// TIA Portal V18 export
FUNCTION_BLOCK "ST10_Flow8_FRobot_2"   // FB1078, GRAPH
// stored: AcknowledgeErrorsRequired false, AutoNumber false, GraphVersion 6.0, InitialValuesAcquisition false, SetENOAutomatically false
   // inherited from GRAPH_BASE
   VAR_INPUT
      INIT_SQ { ExternalAccessible := 'False'; ExternalVisible := 'False'; ExternalWritable := 'False'} : Bool := false;   // Set sequence to initial state
      iSysInface : "RCS_SysComInterface_V1";
   END_VAR
   VAR_IN_OUT
      ioPM_Inface : "RCS_PMInterface_V1";
      ioStatus : Int;
      Auto_Run_after_NG_box_closed : Bool;
   END_VAR
   VAR
      sCtrlMode { S7_SetPoint := 'True'} : "SysFlowCtrlGraph";
      sUpdMES_Data : Bool;   // 更新MES数据
      工件放行中 : Bool;
      前站站号 { ExternalAccessible := 'False'; ExternalVisible := 'False'; ExternalWritable := 'False'} : UInt;
      本站站号 { ExternalAccessible := 'False'; ExternalVisible := 'False'; ExternalWritable := 'False'} : UInt;
      弹窗Temp : Array[1..10] of Int;
      AlarmID : Int;
      TON { S7_SetPoint := 'True'} : Array[0..10] of TON_TIME;
      TOF { S7_SetPoint := 'True'} : Array[0..10] of TOF_TIME;
      sUP { S7_SetPoint := 'True'} : Array[0..10] of Bool;
      更新RFID完成 : Bool;
   END_VAR
   VAR_TEMP
      Tempresult : USInt;
      本站站号乘10 : UInt;
   END_VAR
   VAR CONSTANT
      Gripper_empty : Int := 0;
      "Gripper_have_OK_part_NO-MES" : Int := 199;
      Gripper_have_OK_part : Int := 110;
      Gripper_have_uknown_part : Int := 100;
      Gripper_Product_DMC_not_readable : Int := 155;
   END_VAR
   // // TON[0] : 托盘流入1托盘到位传感器
   // // TON[1] : 托盘流入1托盘到位传感器
   // // TON[2] : 托盘流入1产品有无传感器
   // // TON[3] : 托盘流入1产品有无传感器
   // // TON[4] : 托盘流入1姿态检测光电2
   // // TON[5] : 托盘流入1姿态检测光电3
   // // TON[0].Q : 托盘流入1托盘到位
   // // TON[1].Q : 托盘流入1托盘无
   // // TON[2].Q : 托盘流入1有产品
   // // TON[3].Q : 托盘流入1无产品
   // // TON[4].Q : 托盘流入1姿态检测光电2
   // // TON[5].Q : 托盘流入1姿态检测光电3
BEGIN
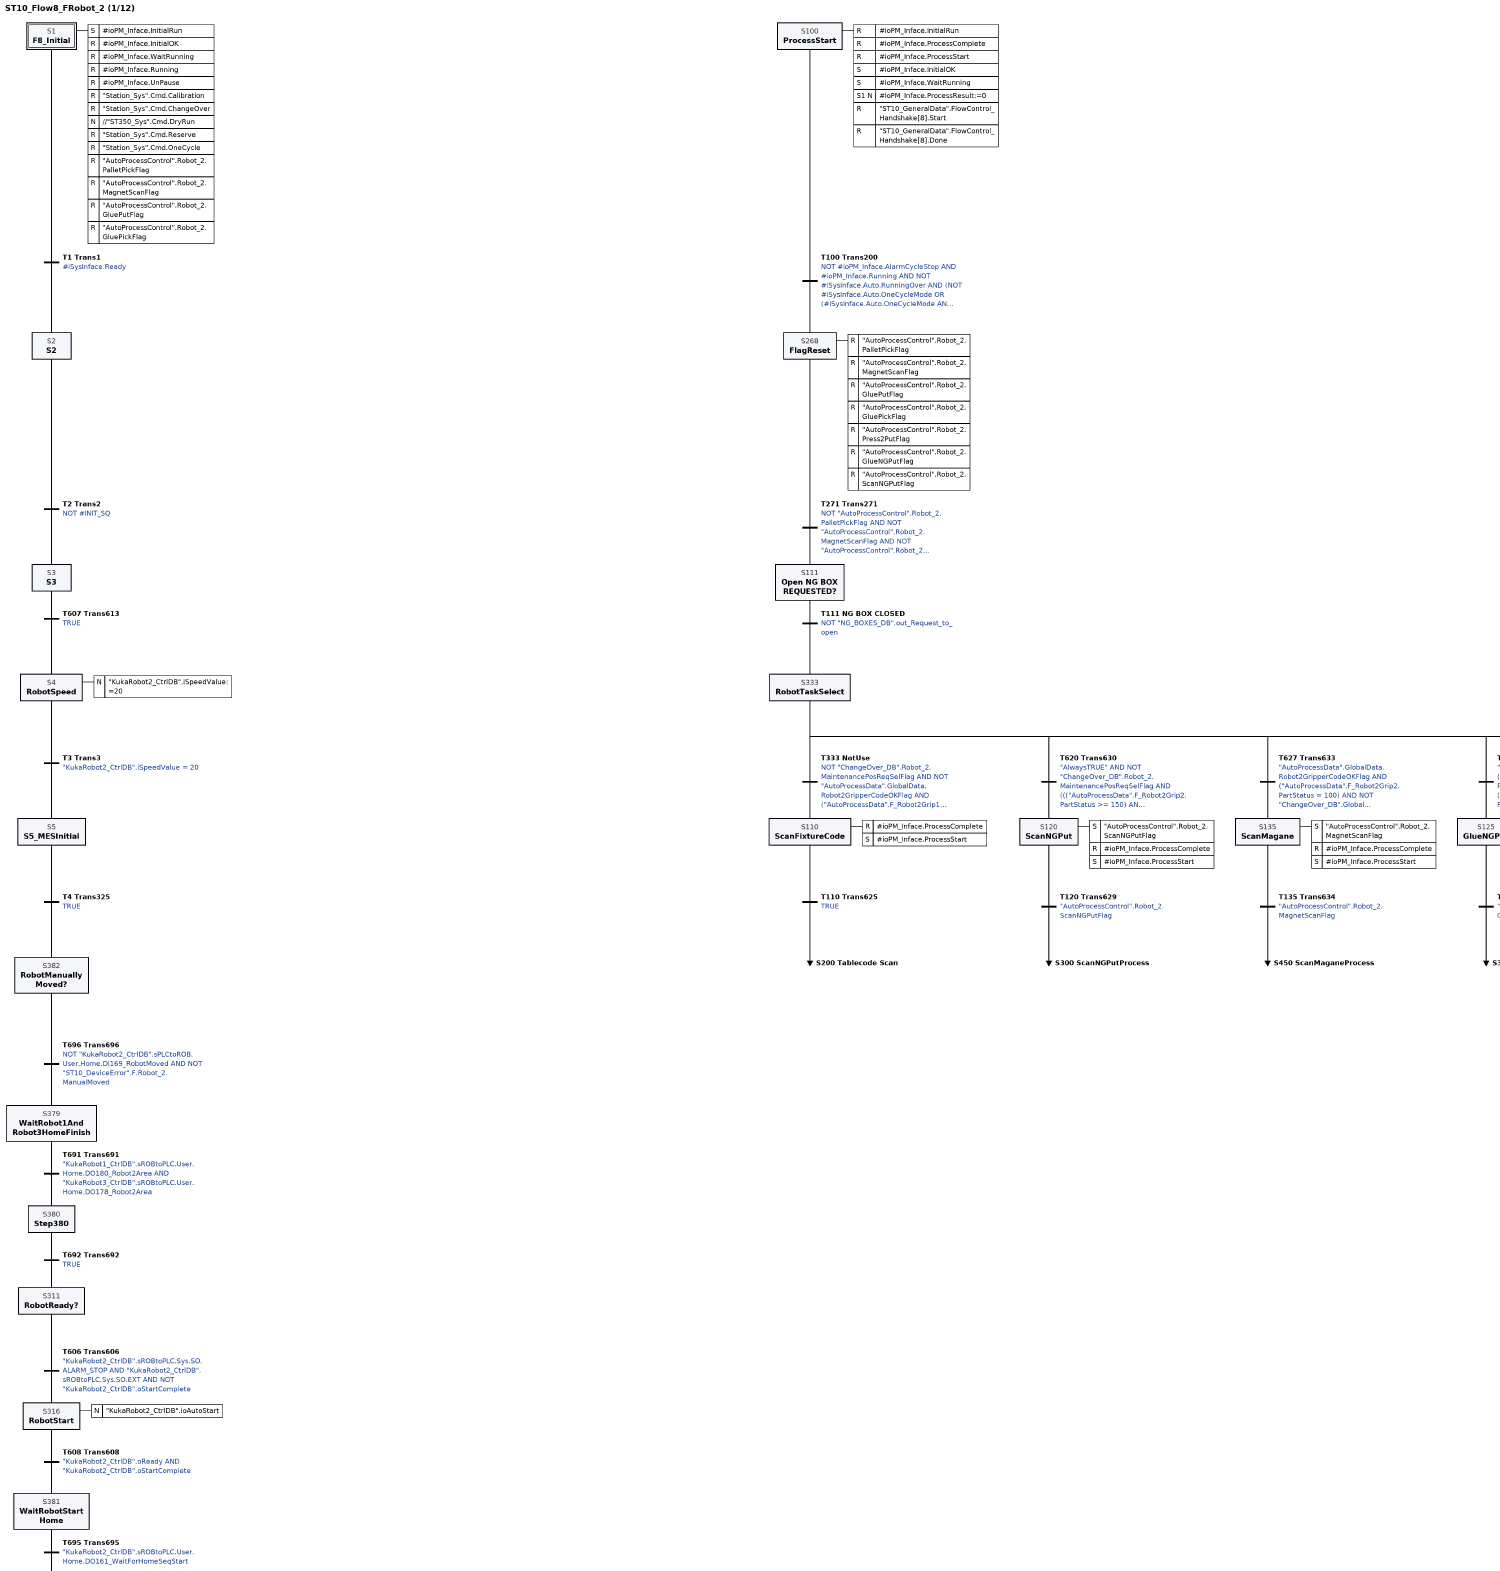
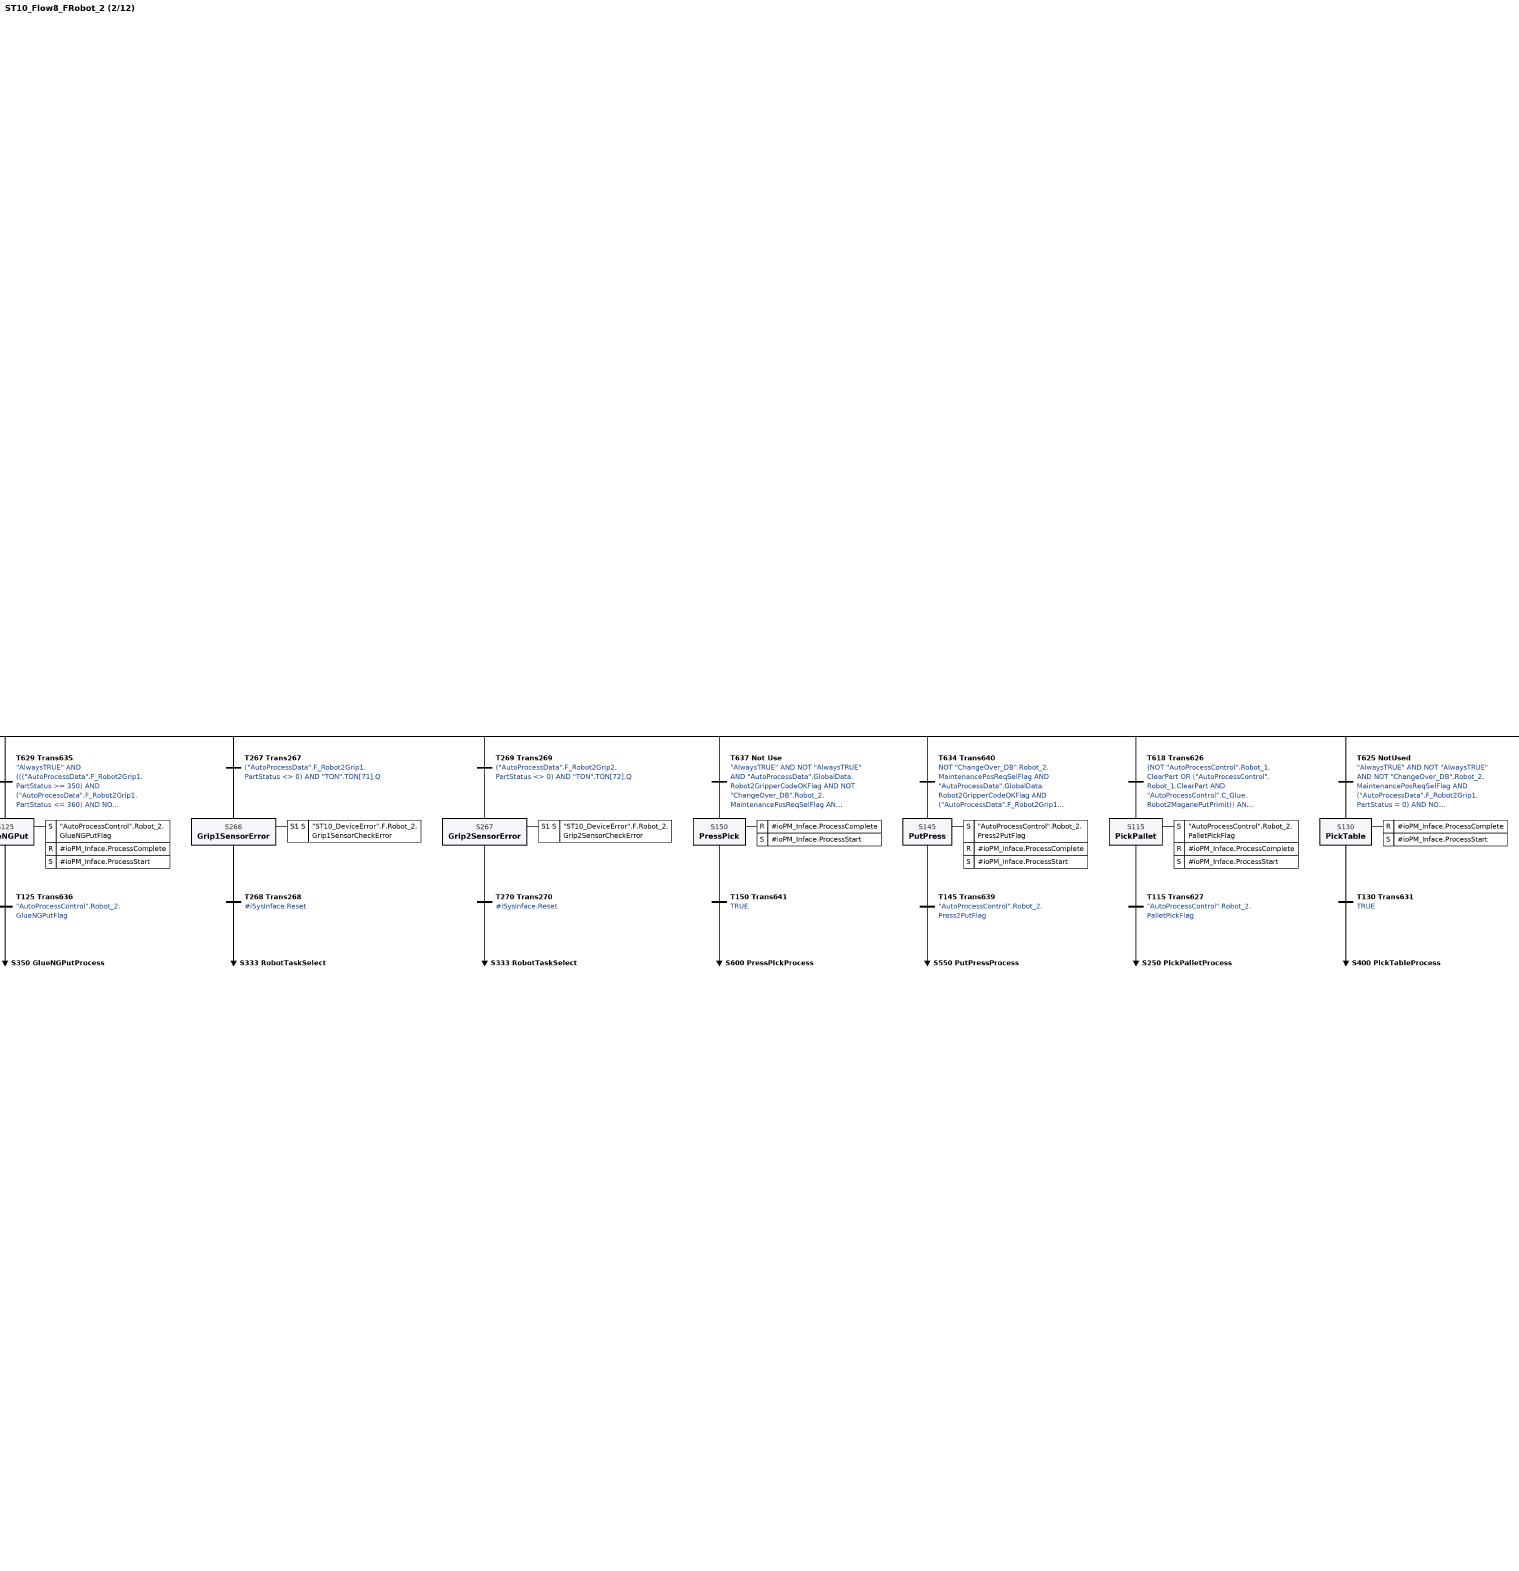
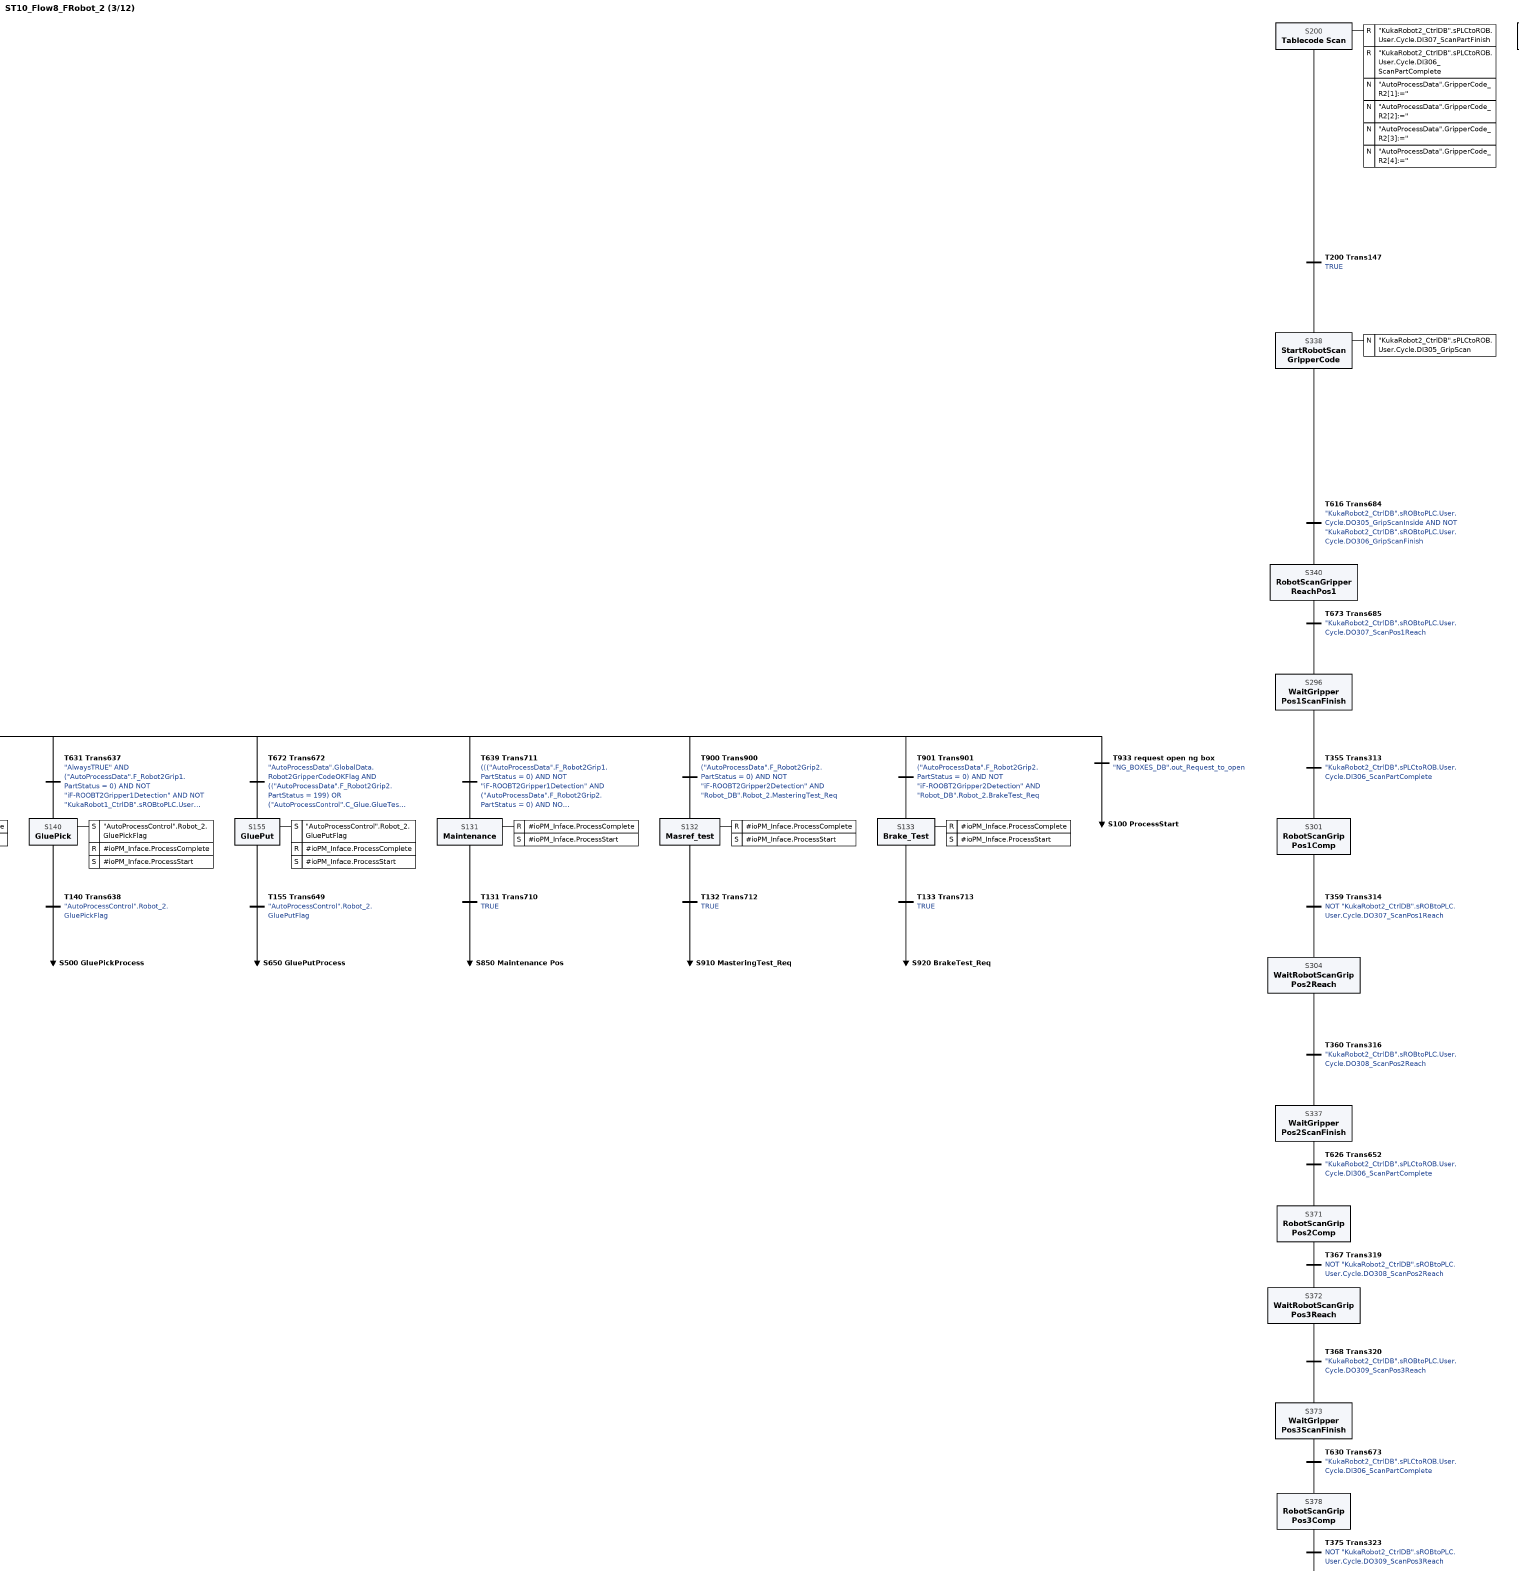
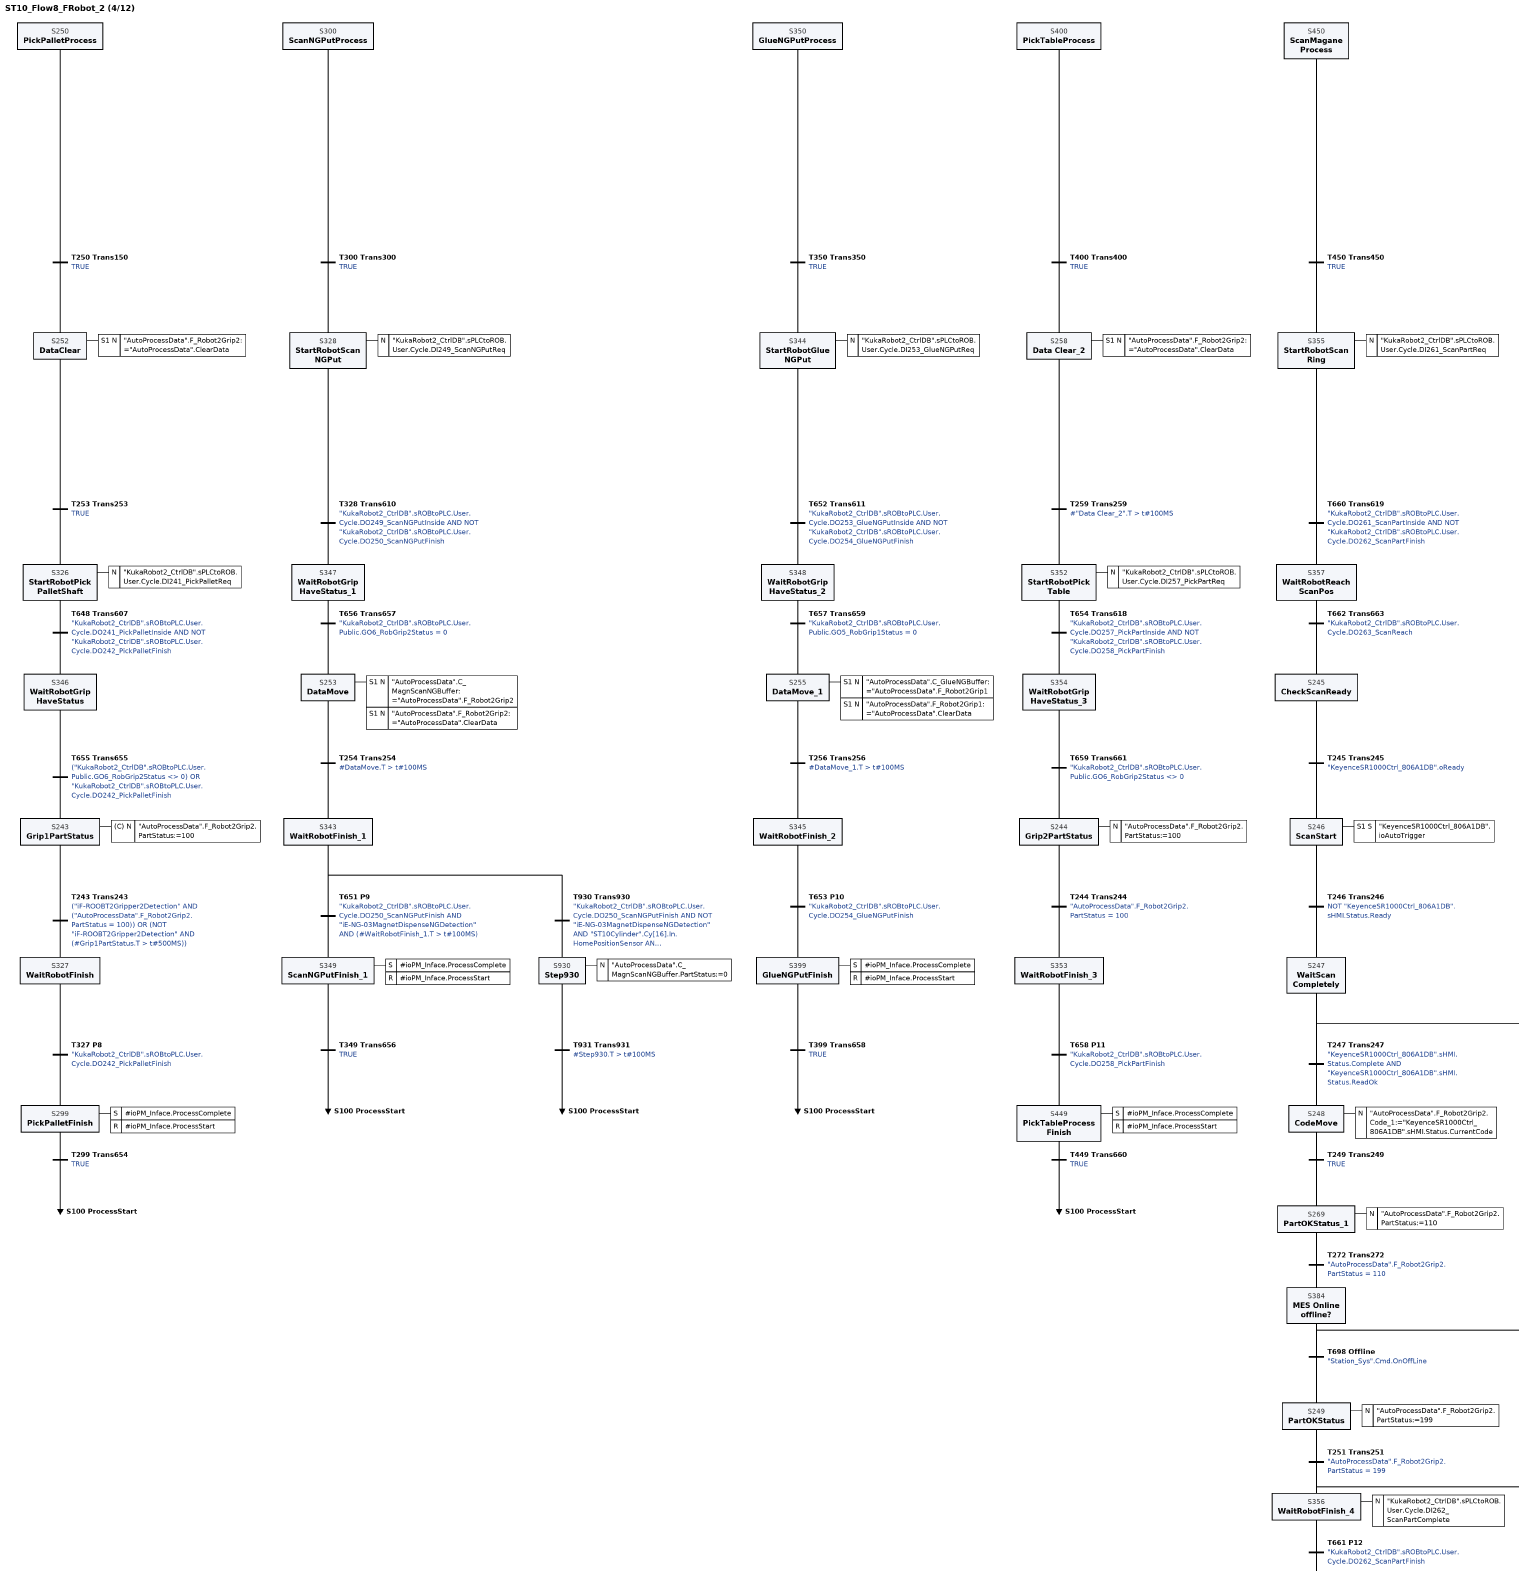
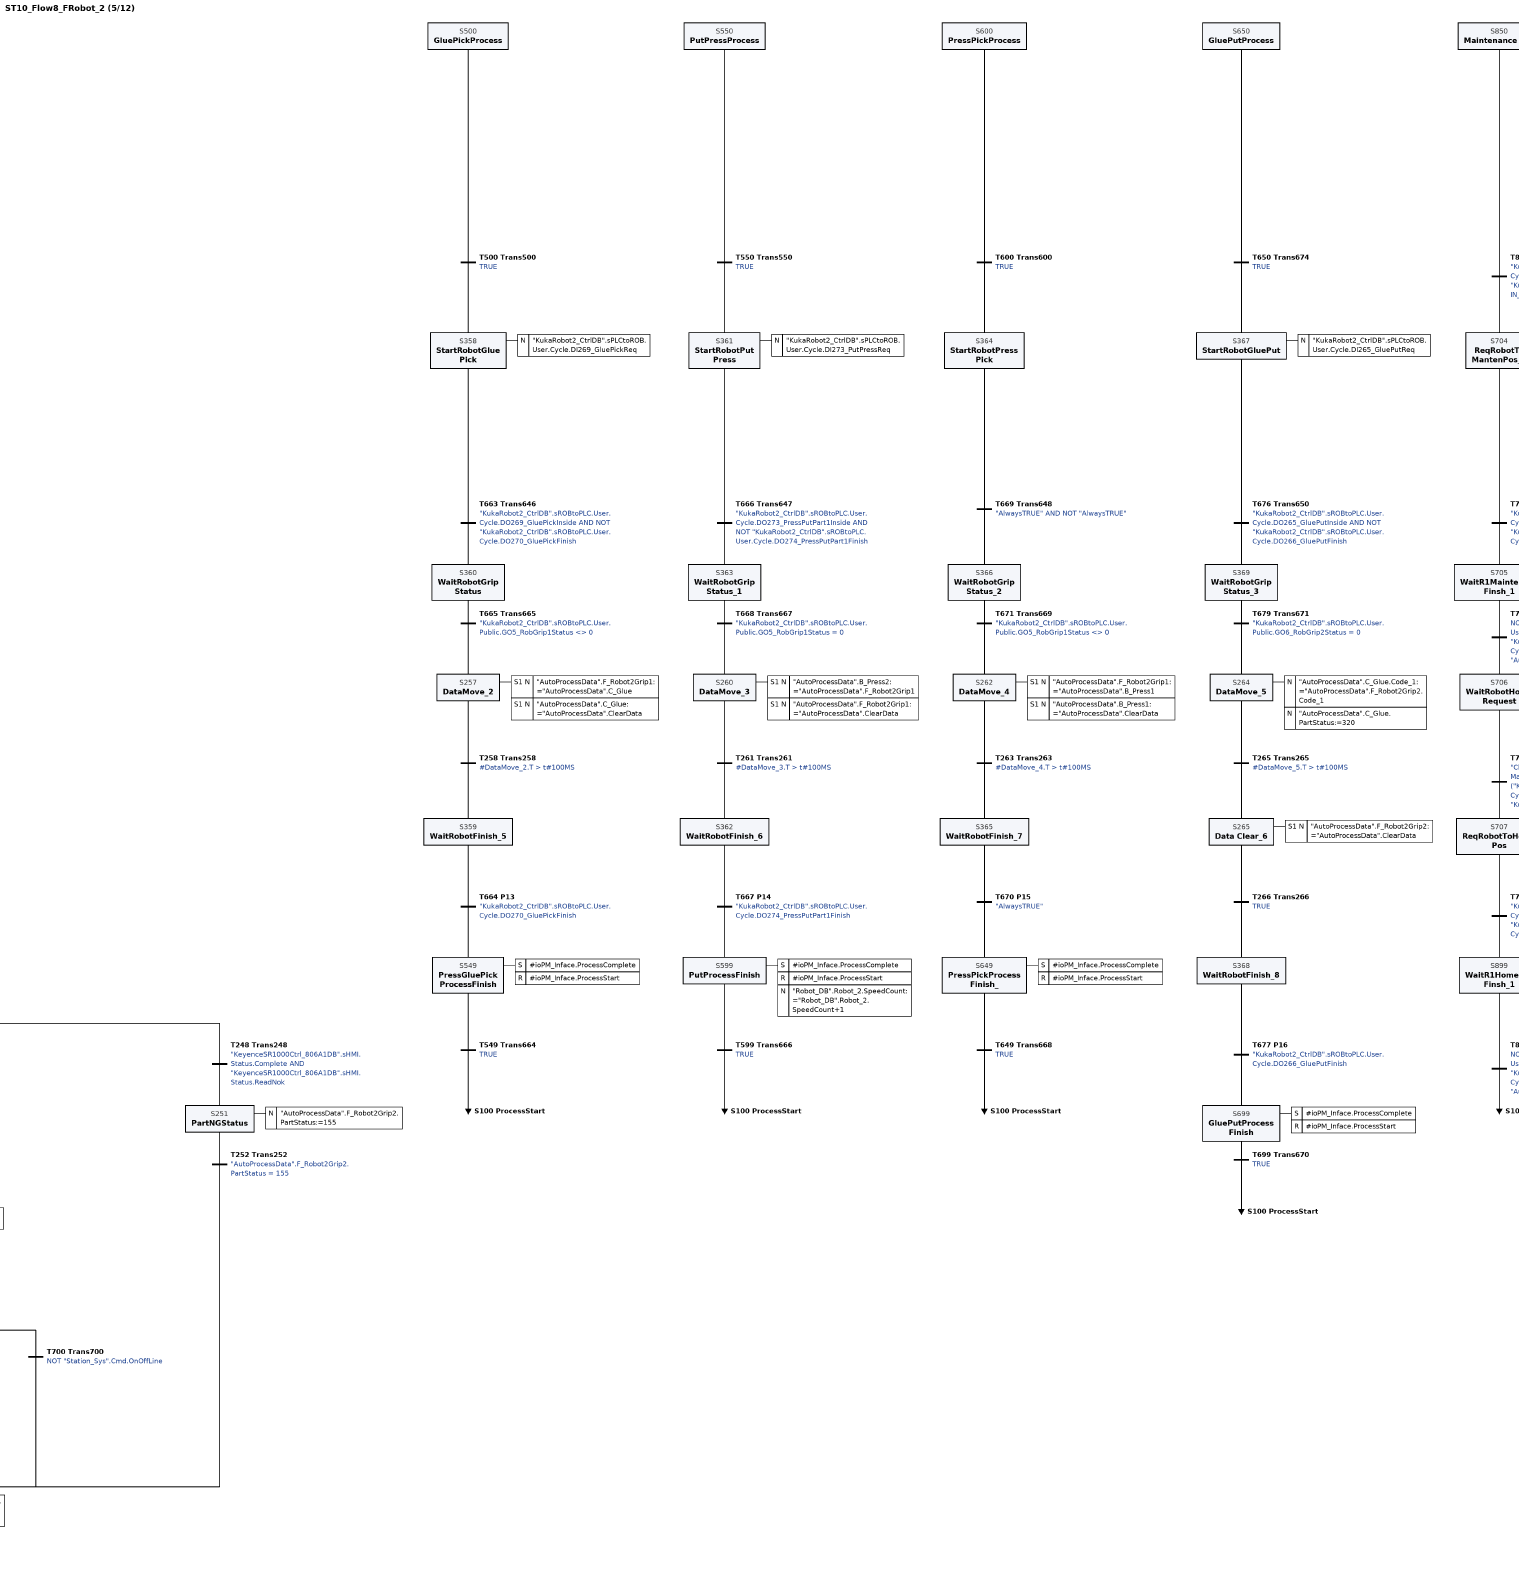
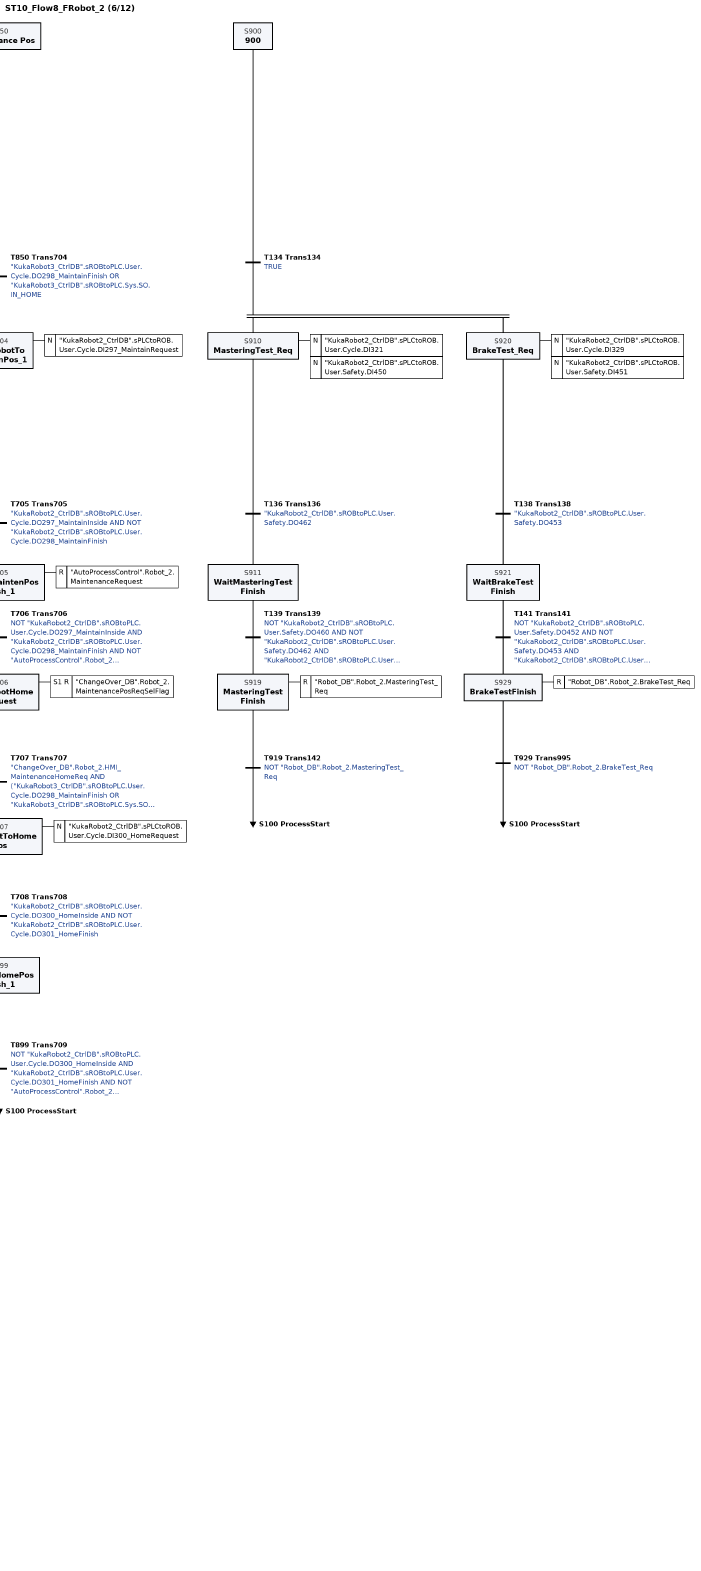
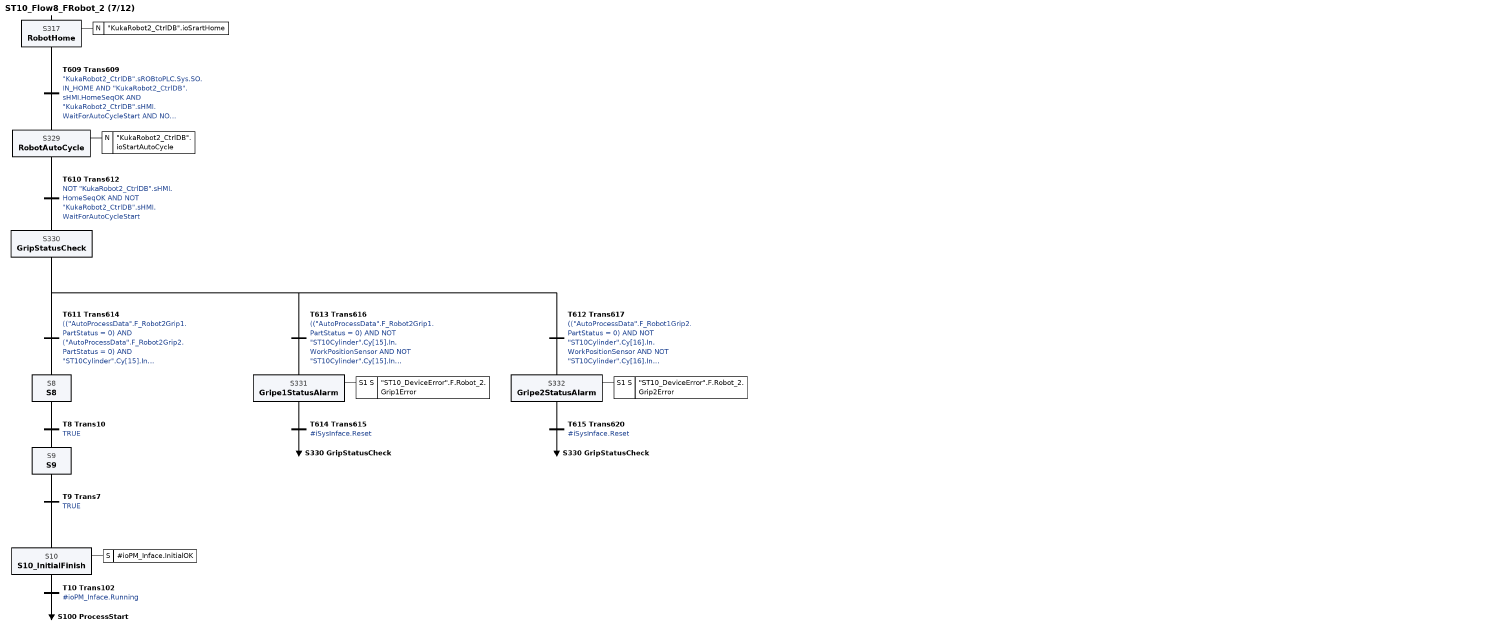
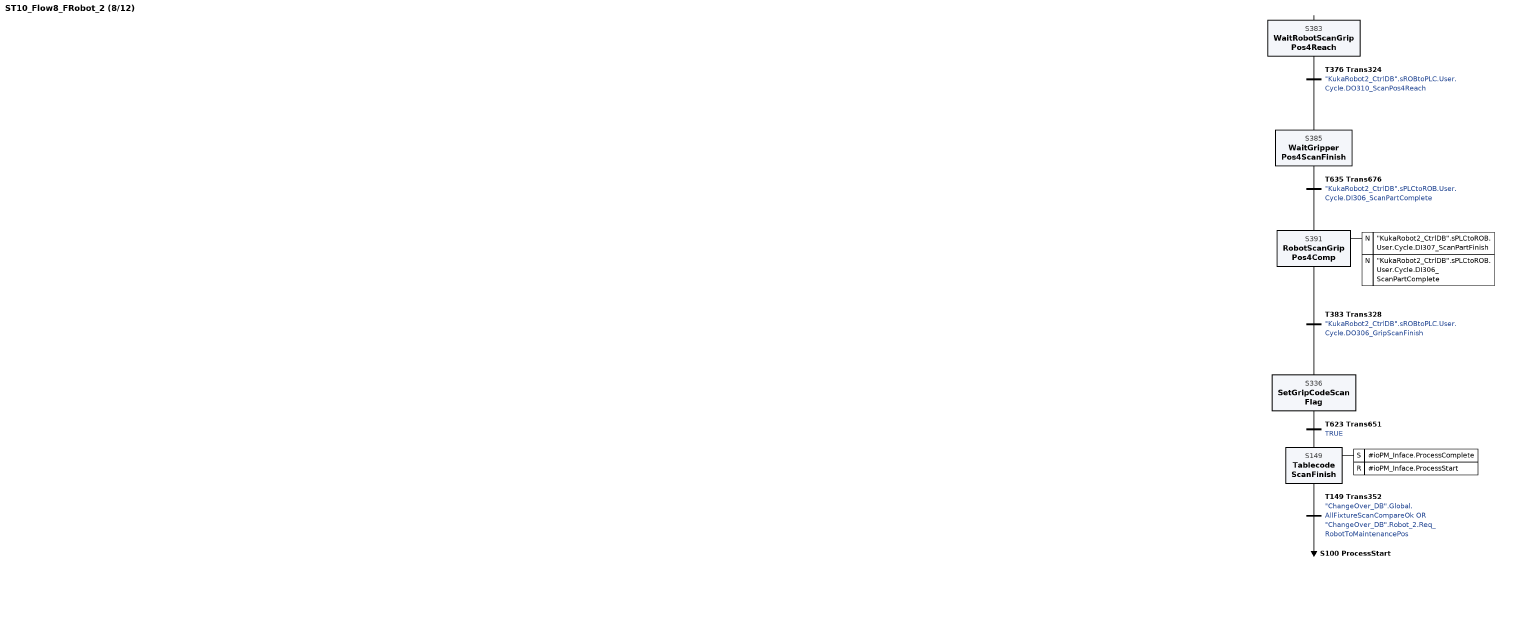
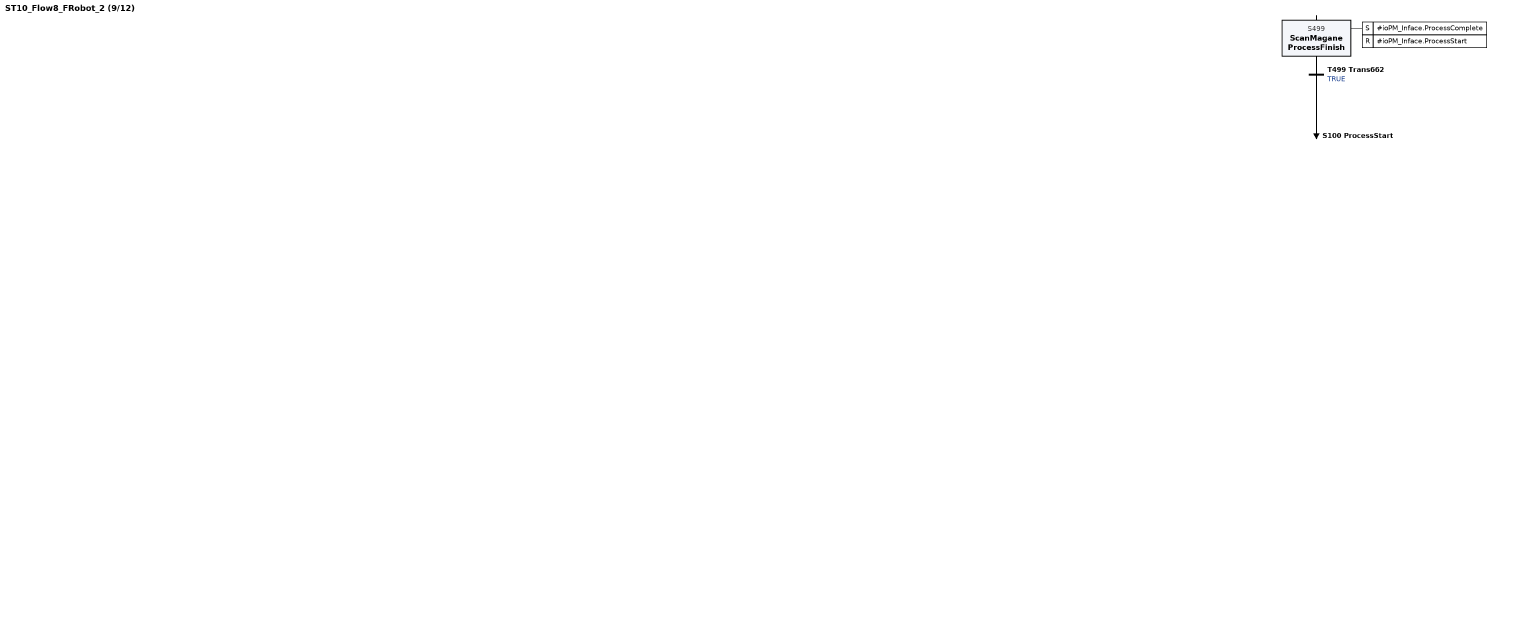
   // permanent pre-instructions
   NETWORK 1
      #TON[10].TON(IN := "AlwaysTRUE" AND "Station_Sys".Alarm.ImmediatelyStop, PT := T#300ms);
      #ioPM_Inface.AlarmImdilyStop := #TON[10].Q;
      #ioPM_Inface.AlarmCycleStop := "AlwaysTRUE" AND "Station_Sys".Alarm.CycleStop;
   NETWORK 2
      IF NOT False THEN
          #sCtrlMode(INIT := #INIT_SQ,   // "SysFlowCtrlGraph"
                     iSysInface := #iSysInface,
                     ioPM_Inface := #ioPM_Inface,
                     ioGraphCtrl := #RT_DATA.MOP);
      END_IF;
   NETWORK 3
      #TON[0].TON(IN := "AlwaysTRUE" AND "iA-Rotating product Check", PT := t#500ms);   // 工位11有托盘
      #TON[1].TOF(IN := "AlwaysTRUE" AND NOT "iA-Rotating product Check", PT := T#300ms);   // 工位无托盘
      #TON[2].TON(IN := "AlwaysTRUE", PT := T#300ms);
      #TON[3].TON(IN := "AlwaysTRUE", PT := T#300ms);
      #TON[4].TON(IN := "AlwaysTRUE", PT := T#300ms);
      #TON[5].TON(IN := "AlwaysTRUE", PT := T#300ms);
   NETWORK 4
      #前站站号 := 345;
      #本站站号 := 350;

   // sequencer 1: S01-S99 初始化 / S01-S99 Initial
   INITIAL_STEP F8_Initial:   // S1, max time T#10S, warning time T#7S
              S    #ioPM_Inface.InitialRun
              R    #ioPM_Inface.InitialOK
              R    #ioPM_Inface.WaitRunning
              R    #ioPM_Inface.Running
              R    #ioPM_Inface.UnPause
              R    "Station_Sys".Cmd.Calibration
              R    "Station_Sys".Cmd.ChangeOver
                   //"ST350_Sys".Cmd.DryRun
              R    "Station_Sys".Cmd.Reserve
              R    "Station_Sys".Cmd.OneCycle
              R    "AutoProcessControl".Robot_2.PalletPickFlag
              R    "AutoProcessControl".Robot_2.MagnetScanFlag
              R    "AutoProcessControl".Robot_2.GluePutFlag
              R    "AutoProcessControl".Robot_2.GluePickFlag
              R    "AutoProcessControl".Robot_2.Press2PutFlag
              R    "AutoProcessControl".Robot_2.GlueNGPutFlag
              R    "AutoProcessControl".Robot_2.ScanNGPutFlag
              R    #ioPM_Inface.ProcessComplete
              R    #ioPM_Inface.ProcessStart
          S1  R    "ChangeOver_DB".Robot_2.MaintenancePosReqSelFlag
                   //"Robot_DB".Robot_2.MasteringTest_Req
                   //"Robot_DB".Robot_2.BrakeTest_Req
          S0  R    #Auto_Run_after_NG_box_closed
   END_STEP
   TRANSITION Trans1 FROM F8_Initial TO S2   // T1
      := #iSysInface.Ready;
   END_TRANSITION
   STEP S2:   // S2, max time T#10S, warning time T#7S
   END_STEP
   TRANSITION Trans2 FROM S2 TO S3   // T2
      := NOT #INIT_SQ;
   END_TRANSITION
   STEP RobotSpeed:   // S4, max time T#10S, warning time T#7S
              N    "KukaRobot2_CtrlDB".iSpeedValue:=20
   END_STEP
   TRANSITION Trans3 FROM RobotSpeed TO S5_MESInitial   // T3
      := "KukaRobot2_CtrlDB".iSpeedValue = 20;
   END_TRANSITION
   STEP S5_MESInitial:   // S5, max time T#10S, warning time T#7S
   END_STEP
   TRANSITION Trans325 FROM S5_MESInitial TO "RobotManuallyMoved?"   // T4
      := TRUE;
   END_TRANSITION
   STEP S10_InitialFinish:   // S10, max time T#10S, warning time T#7S
              S    #ioPM_Inface.InitialOK
   END_STEP
   TRANSITION Trans102 FROM S10_InitialFinish TO ProcessStart   // T10, jump
      := #ioPM_Inface.Running;
   END_TRANSITION
   STEP S3:   // S3, max time T#10S, warning time T#7S
   END_STEP
   TRANSITION Trans613 FROM S3 TO RobotSpeed   // T607
      := TRUE;
   END_TRANSITION
   STEP S8:   // S8, max time T#10S, warning time T#7S
   END_STEP
   TRANSITION Trans10 FROM S8 TO S9   // T8
      := TRUE;
   END_TRANSITION
   STEP S9:   // S9, max time T#10S, warning time T#7S
   END_STEP
   TRANSITION Trans7 FROM S9 TO S10_InitialFinish   // T9
      := TRUE;
   END_TRANSITION
   STEP "RobotReady?":   // S311, max time T#10S, warning time T#7S
   END_STEP
   TRANSITION Trans606 FROM "RobotReady?" TO RobotStart   // T606
      := "KukaRobot2_CtrlDB".sROBtoPLC.Sys.SO.ALARM_STOP AND "KukaRobot2_CtrlDB".sROBtoPLC.Sys.SO.EXT AND NOT "KukaRobot2_CtrlDB".oStartComplete;
   END_TRANSITION
   STEP RobotStart:   // S316, max time T#10S, warning time T#7S
              N    "KukaRobot2_CtrlDB".ioAutoStart
   END_STEP
   TRANSITION Trans608 FROM RobotStart TO WaitRobotStartHome   // T608
      := "KukaRobot2_CtrlDB".oReady AND "KukaRobot2_CtrlDB".oStartComplete;
   END_TRANSITION
   STEP RobotHome:   // S317, max time T#10S, warning time T#7S
              N    "KukaRobot2_CtrlDB".ioSrartHome
   END_STEP
   TRANSITION Trans609 FROM RobotHome TO RobotAutoCycle   // T609
      := "KukaRobot2_CtrlDB".sROBtoPLC.Sys.SO.IN_HOME AND "KukaRobot2_CtrlDB".sHMI.HomeSeqOK AND "KukaRobot2_CtrlDB".sHMI.WaitForAutoCycleStart AND NOT "KukaRobot2_CtrlDB".sHMI.GoHomeFail;
   END_TRANSITION
   STEP RobotAutoCycle:   // S329, max time T#10S, warning time T#7S
              N    "KukaRobot2_CtrlDB".ioStartAutoCycle
   END_STEP
   TRANSITION Trans612 FROM RobotAutoCycle TO GripStatusCheck   // T610
      := NOT "KukaRobot2_CtrlDB".sHMI.HomeSeqOK AND NOT "KukaRobot2_CtrlDB".sHMI.WaitForAutoCycleStart;
   END_TRANSITION
   STEP GripStatusCheck:   // S330, max time T#10S, warning time T#7S
   END_STEP
   TRANSITION Trans614 FROM GripStatusCheck TO S8   // T611
      := (("AutoProcessData".F_Robot2Grip1.PartStatus = 0) AND ("AutoProcessData".F_Robot2Grip2.PartStatus = 0) AND "ST10Cylinder".Cy[15].In.HomePositionSensor AND "ST10Cylinder".Cy[16].In.HomePositionSensor) OR (("AutoProcessData".F_Robot2Grip1.PartStatus <> 0) AND NOT "ST10Cylinder".Cy[15].In.WorkPositionSensor AND NOT "ST10Cylinder".Cy[15].In.HomePositionSensor) OR (("AutoProcessData".F_Robot2Grip2.PartStatus <> 0) AND NOT "ST10Cylinder".Cy[16].In.WorkPositionSensor AND NOT "ST10Cylinder".Cy[16].In.HomePositionSensor);
   END_TRANSITION
   TRANSITION Trans616 FROM GripStatusCheck TO Gripe1StatusAlarm   // T613
      := (("AutoProcessData".F_Robot2Grip1.PartStatus = 0) AND NOT "ST10Cylinder".Cy[15].In.WorkPositionSensor AND NOT "ST10Cylinder".Cy[15].In.HomePositionSensor) OR (("AutoProcessData".F_Robot2Grip1.PartStatus <> 0) AND "ST10Cylinder".Cy[15].In.WorkPositionSensor);
   END_TRANSITION
   TRANSITION Trans617 FROM GripStatusCheck TO Gripe2StatusAlarm   // T612
      := (("AutoProcessData".F_Robot1Grip2.PartStatus = 0) AND NOT "ST10Cylinder".Cy[16].In.WorkPositionSensor AND NOT "ST10Cylinder".Cy[16].In.HomePositionSensor) OR (("AutoProcessData".F_Robot1Grip2.PartStatus <> 0) AND "ST10Cylinder".Cy[16].In.WorkPositionSensor);
   END_TRANSITION
   STEP Gripe1StatusAlarm:   // S331, max time T#10S, warning time T#7S
          S1  S    "ST10_DeviceError".F.Robot_2.Grip1Error
   END_STEP
   TRANSITION Trans615 FROM Gripe1StatusAlarm TO GripStatusCheck   // T614, jump
      := #iSysInface.Reset;
   END_TRANSITION
   STEP Gripe2StatusAlarm:   // S332, max time T#10S, warning time T#7S
          S1  S    "ST10_DeviceError".F.Robot_2.Grip2Error
   END_STEP
   TRANSITION Trans620 FROM Gripe2StatusAlarm TO GripStatusCheck   // T615, jump
      := #iSysInface.Reset;
   END_TRANSITION
   STEP WaitRobot1AndRobot3HomeFinish:   // S379, max time T#10S, warning time T#7S
   END_STEP
   TRANSITION Trans691 FROM WaitRobot1AndRobot3HomeFinish TO Step380   // T691
      := "KukaRobot1_CtrlDB".sROBtoPLC.User.Home.DO180_Robot2Area AND "KukaRobot3_CtrlDB".sROBtoPLC.User.Home.DO178_Robot2Area;
   END_TRANSITION
   STEP Step380:   // S380, max time T#10S, warning time T#7S
   END_STEP
   TRANSITION Trans692 FROM Step380 TO "RobotReady?"   // T692
      := TRUE;
   END_TRANSITION
   STEP WaitRobotStartHome:   // S381, max time T#10S, warning time T#7S
   END_STEP
   TRANSITION Trans695 FROM WaitRobotStartHome TO RobotHome   // T695
      := "KukaRobot2_CtrlDB".sROBtoPLC.User.Home.DO161_WaitForHomeSeqStart;
   END_TRANSITION
   STEP "RobotManuallyMoved?":   // S382, max time T#10S, warning time T#7S
   END_STEP
   TRANSITION Trans696 FROM "RobotManuallyMoved?" TO WaitRobot1AndRobot3HomeFinish   // T696
      := NOT "KukaRobot2_CtrlDB".sPLCtoROB.User.Home.DI169_RobotMoved AND NOT "ST10_DeviceError".F.Robot_2.ManualMoved;
   END_TRANSITION

   // sequencer 2: S100-S199 等待到位 / S100-S199 RobotTask
   STEP ProcessStart:   // S100, max time T#10S, warning time T#7S
      // 自动等待开始运行
              R    #ioPM_Inface.InitialRun
              R    #ioPM_Inface.ProcessComplete
              R    #ioPM_Inface.ProcessStart
              S    #ioPM_Inface.InitialOK
              S    #ioPM_Inface.WaitRunning
          S1  N    #ioPM_Inface.ProcessResult:=0
              R    "ST10_GeneralData".FlowControl_Handshake[8].Start
              R    "ST10_GeneralData".FlowControl_Handshake[8].Done
   END_STEP
   TRANSITION Trans200 FROM ProcessStart TO FlagReset   // T100
      := NOT #ioPM_Inface.AlarmCycleStop AND #ioPM_Inface.Running AND NOT #iSysInface.Auto.RunningOver AND (NOT #iSysInface.Auto.OneCycleMode OR (#iSysInface.Auto.OneCycleMode AND #ioPM_Inface.TriggerOneCycle));
   END_TRANSITION
   STEP ScanFixtureCode:   // S110, max time T#10S, warning time T#7S
              R    #ioPM_Inface.ProcessComplete
              S    #ioPM_Inface.ProcessStart
   END_STEP
   TRANSITION Trans625 FROM ScanFixtureCode TO "Tablecode Scan"   // T110, jump
      := TRUE;
   END_TRANSITION
   STEP RobotTaskSelect:   // S333, max time T#10S, warning time T#7S
   END_STEP
   TRANSITION NotUse FROM RobotTaskSelect TO ScanFixtureCode   // T333
      := NOT "ChangeOver_DB".Robot_2.MaintenancePosReqSelFlag AND NOT "AutoProcessData".GlobalData.Robot2GripperCodeOKFlag AND ("AutoProcessData".F_Robot2Grip1.PartStatus = 0) AND NOT "iF-ROOBT2Gripper1Detection" AND "AutoProcessControl".Robot_2.GripScanRequest AND NOT "KukaRobot1_CtrlDB".sROBtoPLC.User.Cycle.DO297_MaintainInside AND NOT "ChangeOver_DB".Robot_1.MaintenancePosReqSelFlag AND NOT "Robot_DB".Robot_2.MasteringTest_Req AND NOT "Robot_DB".Robot_2.BrakeTest_Req;
   END_TRANSITION
   TRANSITION Trans630 FROM RobotTaskSelect TO ScanNGPut   // T620
      := "AlwaysTRUE" AND NOT "ChangeOver_DB".Robot_2.MaintenancePosReqSelFlag AND ((("AutoProcessData".F_Robot2Grip2.PartStatus >= 150) AND ("AutoProcessData".F_Robot2Grip2.PartStatus <= 160)) OR (("AutoProcessData".F_Robot2Grip2.PartStatus = 0) AND NOT "ST10Cylinder".Cy[16].In.HomePositionSensor AND NOT "ST10Cylinder".Cy[16].In.WorkPositionSensor) OR (("AutoProcessData".F_Robot2Grip2.PartStatus >= 155) AND "ST10Cylinder".Cy[16].In.WorkPositionSensor)) AND NOT "iE-NG-03MagnetDispenseNGDetection" AND "KukaRobot3_CtrlDB".sROBtoPLC.User.Home.DO178_Robot2Area AND NOT "KukaRobot3_CtrlDB".sROBtoPLC.User.Cycle.DO253_PickGlueNGInside AND NOT "KukaRobot3_CtrlDB".sROBtoPLC.User.Cycle.DO249_PickMagnetInside AND NOT "KukaRobot3_CtrlDB".sROBtoPLC.User.Cycle.DO277_PressPutRingInside AND NOT "AutoProcessControl".Robot_3.Press2PickFlag AND NOT "AutoProcessControl".Robot_3.GlueNGPickFlag AND NOT "AutoProcessControl".Robot_3.ScanNGPickFlag AND ("AutoProcessControl".Robot2ScanNG.PutPrimit OR NOT "iE-NG-03MagnetDispenseNGDetection") AND NOT "KukaRobot1_CtrlDB".sROBtoPLC.User.Cycle.DO297_MaintainInside AND NOT "ChangeOver_DB".Robot_1.MaintenancePosReqSelFlag;
   END_TRANSITION
   TRANSITION Trans633 FROM RobotTaskSelect TO ScanMagane   // T627
      := "AutoProcessData".GlobalData.Robot2GripperCodeOKFlag AND ("AutoProcessData".F_Robot2Grip2.PartStatus = 100) AND NOT "ChangeOver_DB".Global.ManualModeFlag AND ("iF-ROOBT2Gripper2Detection" OR "AlwaysTRUE") AND NOT "ST10Cylinder".Cy[16].In.HomePositionSensor AND "KukaRobot1_CtrlDB".sROBtoPLC.User.Home.DO180_Robot2Area AND NOT "KukaRobot1_CtrlDB".sROBtoPLC.User.Cycle.DO289_GluePutInside AND NOT "ChangeOver_DB".Robot_2.MaintenancePosReqSelFlag AND NOT "KukaRobot1_CtrlDB".sROBtoPLC.User.Cycle.DO297_MaintainInside AND NOT "ChangeOver_DB".Robot_1.MaintenancePosReqSelFlag AND NOT "Robot_DB".Robot_2.MasteringTest_Req AND NOT "Robot_DB".Robot_2.BrakeTest_Req;
   END_TRANSITION
   TRANSITION Trans635 FROM RobotTaskSelect TO GlueNGPut   // T629
      := "AlwaysTRUE" AND ((("AutoProcessData".F_Robot2Grip1.PartStatus >= 350) AND ("AutoProcessData".F_Robot2Grip1.PartStatus <= 360) AND NOT "iF-ROOBT2Gripper1Detection") OR ("AutoProcessControl".C_Glue.GlueTest AND ("AutoProcessData".F_Robot2Grip1.PartStatus = 399))) AND NOT "ST10Cylinder".Cy[15].In.HomePositionSensor AND NOT "iE-NG-03ShaftDispenseNGDetection" AND NOT "ChangeOver_DB".Robot_2.MaintenancePosReqSelFlag AND "KukaRobot3_CtrlDB".sROBtoPLC.User.Home.DO178_Robot2Area AND NOT "KukaRobot3_CtrlDB".sROBtoPLC.User.Cycle.DO253_PickGlueNGInside AND NOT "KukaRobot3_CtrlDB".sROBtoPLC.User.Cycle.DO249_PickMagnetInside AND NOT "KukaRobot3_CtrlDB".sROBtoPLC.User.Cycle.DO277_PressPutRingInside AND NOT "AutoProcessControl".Robot_3.Press2PickFlag AND NOT "AutoProcessControl".Robot_3.GlueNGPickFlag AND NOT "AutoProcessControl".Robot_3.ScanNGPickFlag AND ("AutoProcessControl".Robot2GlueNG.PutPrimit OR ("AutoProcessControl".C_Glue.GlueTest AND NOT "AutoProcessControl".Robot2GlueNG.PutPrimit)) AND NOT "KukaRobot1_CtrlDB".sROBtoPLC.User.Cycle.DO297_MaintainInside AND NOT "ChangeOver_DB".Robot_1.MaintenancePosReqSelFlag;
   END_TRANSITION
   TRANSITION Trans267 FROM RobotTaskSelect TO Grip1SensorError   // T267
      := ("AutoProcessData".F_Robot2Grip1.PartStatus <> 0) AND "TON".TON[71].Q;
   END_TRANSITION
   TRANSITION Trans269 FROM RobotTaskSelect TO Grip2SensorError   // T269
      := ("AutoProcessData".F_Robot2Grip2.PartStatus <> 0) AND "TON".TON[72].Q;
   END_TRANSITION
   TRANSITION "Not Use" FROM RobotTaskSelect TO PressPick   // T637
      := "AlwaysTRUE" AND NOT "AlwaysTRUE" AND "AutoProcessData".GlobalData.Robot2GripperCodeOKFlag AND NOT "ChangeOver_DB".Robot_2.MaintenancePosReqSelFlag AND ("AutoProcessData".F_Robot2Grip1.PartStatus = 0) AND NOT "iF-ROOBT2Gripper1Detection" AND "ST10Cylinder".Cy[15].In.HomePositionSensor AND "AutoProcessControl".B_Press_1.Robot1PickPrimit AND NOT "Robot_DB".Robot_2.MasteringTest_Req AND NOT "Robot_DB".Robot_2.BrakeTest_Req;
   END_TRANSITION
   TRANSITION Trans640 FROM RobotTaskSelect TO PutPress   // T634
      := NOT "ChangeOver_DB".Robot_2.MaintenancePosReqSelFlag AND "AutoProcessData".GlobalData.Robot2GripperCodeOKFlag AND ("AutoProcessData".F_Robot2Grip1.PartStatus = 399) AND NOT "ChangeOver_DB".Global.ManualModeFlag AND ("iF-ROOBT2Gripper1Detection" OR "AlwaysTRUE") AND NOT "ST10Cylinder".Cy[15].In.HomePositionSensor AND NOT "KukaRobot3_CtrlDB".sROBtoPLC.User.Cycle.DO253_PickGlueNGInside AND NOT "KukaRobot3_CtrlDB".sROBtoPLC.User.Cycle.DO249_PickMagnetInside AND NOT "KukaRobot3_CtrlDB".sROBtoPLC.User.Cycle.DO277_PressPutRingInside AND "KukaRobot3_CtrlDB".sROBtoPLC.User.Home.DO177_PressPut1Area AND "KukaRobot3_CtrlDB".sROBtoPLC.User.Home.DO178_Robot2Area AND NOT "AutoProcessControl".Robot_3.Press2PickFlag AND NOT "AutoProcessControl".Robot_3.GlueNGPickFlag AND NOT "AutoProcessControl".Robot_3.ScanNGPickFlag AND "AutoProcessControl".B_Press_2.Robot2PutPrimit AND NOT "Robot_DB".Robot_2.MasteringTest_Req AND NOT "Robot_DB".Robot_2.BrakeTest_Req;
   END_TRANSITION
   TRANSITION Trans626 FROM RobotTaskSelect TO PickPallet   // T618
      := (NOT "AutoProcessControl".Robot_1.ClearPart OR ("AutoProcessControl".Robot_1.ClearPart AND "AutoProcessControl".C_Glue.Robot2MaganePutPrimit)) AND "AutoProcessData".GlobalData.Robot2GripperCodeOKFlag AND NOT "ChangeOver_DB".Global.ScanFixtureFlag AND NOT "ChangeOver_DB".Global.ManualModeFlag AND ("AutoProcessData".F_Robot2Grip2.PartStatus = 0) AND NOT "iF-ROOBT2Gripper2Detection" AND ("AutoProcessData".F_Robot2Grip1.PartStatus = 0) AND NOT "iF-ROOBT2Gripper1Detection" AND ("AutoProcessData".C_Glue.PartStatus <> 0) AND "KukaRobot1_CtrlDB".sROBtoPLC.User.Home.DO179_GlueArea AND "KukaRobot1_CtrlDB".sROBtoPLC.User.Home.DO180_Robot2Area AND NOT "KukaRobot1_CtrlDB".sROBtoPLC.User.Cycle.DO289_GluePutInside AND NOT "AutoProcessControl".Robot_1.GluePutFlag AND NOT "AutoProcessControl".Global.J.EmptyPallet AND NOT "AutoProcessControl".C_Glue.Robot2PickPrimit AND "AutoProcessControl".J_MagnetLine.Robot2PickPrimit AND NOT "ChangeOver_DB".Robot_2.MaintenancePosReqSelFlag AND NOT "KukaRobot1_CtrlDB".sROBtoPLC.User.Cycle.DO297_MaintainInside AND NOT "ChangeOver_DB".Robot_1.MaintenancePosReqSelFlag AND NOT "Robot_DB".Robot_2.MasteringTest_Req AND NOT "Robot_DB".Robot_2.BrakeTest_Req;
   END_TRANSITION
   TRANSITION NotUsed FROM RobotTaskSelect TO PickTable   // T625
      := "AlwaysTRUE" AND NOT "AlwaysTRUE" AND NOT "ChangeOver_DB".Robot_2.MaintenancePosReqSelFlag AND ("AutoProcessData".F_Robot2Grip1.PartStatus = 0) AND NOT "iF-ROOBT2Gripper1Detection" AND "ST10Cylinder".Cy[15].In.HomePositionSensor AND ("AutoProcessData".F_Robot2Grip2.PartStatus = 0) AND NOT "iF-ROOBT2Gripper2Detection" AND "ST10Cylinder".Cy[16].In.HomePositionSensor AND NOT "Robot_DB".Robot_2.MasteringTest_Req AND NOT "Robot_DB".Robot_2.BrakeTest_Req;
   END_TRANSITION
   TRANSITION Trans637 FROM RobotTaskSelect TO GluePick   // T631
      := "AlwaysTRUE" AND ("AutoProcessData".F_Robot2Grip1.PartStatus = 0) AND NOT "iF-ROOBT2Gripper1Detection" AND NOT "KukaRobot1_CtrlDB".sROBtoPLC.User.Cycle.DO289_GluePutInside AND "KukaRobot1_CtrlDB".sROBtoPLC.User.Home.DO180_Robot2Area AND NOT "AutoProcessControl".Robot_1.GluePutFlag AND "AutoProcessControl".C_Glue.Robot2PickPrimit AND NOT "ChangeOver_DB".Robot_2.MaintenancePosReqSelFlag AND NOT "KukaRobot1_CtrlDB".sROBtoPLC.User.Cycle.DO297_MaintainInside AND NOT "ChangeOver_DB".Robot_1.MaintenancePosReqSelFlag AND NOT "Robot_DB".Robot_2.MasteringTest_Req AND NOT "Robot_DB".Robot_2.BrakeTest_Req;
   END_TRANSITION
   TRANSITION Trans672 FROM RobotTaskSelect TO GluePut   // T672
      := "AutoProcessData".GlobalData.Robot2GripperCodeOKFlag AND (("AutoProcessData".F_Robot2Grip2.PartStatus = 199) OR ("AutoProcessControl".C_Glue.GlueTest AND (("AutoProcessData".F_Robot2Grip2.PartStatus = 150) OR ("AutoProcessData".F_Robot2Grip2.PartStatus = 199)))) AND ("iF-ROOBT2Gripper2Detection" OR "AlwaysTRUE") AND NOT "ST10Cylinder".Cy[16].In.HomePositionSensor AND NOT "KukaRobot1_CtrlDB".sROBtoPLC.User.Cycle.DO289_GluePutInside AND "KukaRobot1_CtrlDB".sROBtoPLC.User.Home.DO180_Robot2Area AND NOT "AutoProcessControl".Robot_1.GluePutFlag AND "AutoProcessControl".C_Glue.Robot2MaganePutPrimit AND NOT "ChangeOver_DB".Robot_2.MaintenancePosReqSelFlag AND NOT "KukaRobot1_CtrlDB".sROBtoPLC.User.Cycle.DO297_MaintainInside AND NOT "ChangeOver_DB".Robot_1.MaintenancePosReqSelFlag;
   END_TRANSITION
   TRANSITION Trans711 FROM RobotTaskSelect TO Maintenance   // T639
      := ((("AutoProcessData".F_Robot2Grip1.PartStatus = 0) AND NOT "iF-ROOBT2Gripper1Detection" AND ("AutoProcessData".F_Robot2Grip2.PartStatus = 0) AND NOT "iF-ROOBT2Gripper2Detection" AND "ChangeOver_DB".Robot_2.Req_RobotToMaintenancePos) OR (NOT "AutoProcessControl".Robot_2.MaintenanceRequest AND "ChangeOver_DB".Robot_2.HMI_MaintenancePosActive)) AND NOT "Robot_DB".Robot_2.MasteringTest_Req AND NOT "Robot_DB".Robot_2.BrakeTest_Req;
   END_TRANSITION
   TRANSITION Trans900 FROM RobotTaskSelect TO Masref_test   // T900
      := ("AutoProcessData".F_Robot2Grip2.PartStatus = 0) AND NOT "iF-ROOBT2Gripper2Detection" AND "Robot_DB".Robot_2.MasteringTest_Req;
   END_TRANSITION
   TRANSITION Trans901 FROM RobotTaskSelect TO Brake_Test   // T901
      := ("AutoProcessData".F_Robot2Grip2.PartStatus = 0) AND NOT "iF-ROOBT2Gripper2Detection" AND "Robot_DB".Robot_2.BrakeTest_Req;
   END_TRANSITION
   TRANSITION "request open ng box" FROM RobotTaskSelect TO ProcessStart   // T933, jump
      := "NG_BOXES_DB".out_Request_to_open;
   END_TRANSITION
   STEP PickTable:   // S130, max time T#10S, warning time T#7S
              R    #ioPM_Inface.ProcessComplete
              S    #ioPM_Inface.ProcessStart
   END_STEP
   TRANSITION Trans631 FROM PickTable TO PickTableProcess   // T130, jump
      := TRUE;
   END_TRANSITION
   STEP ScanNGPut:   // S120, max time T#10S, warning time T#7S
              S    "AutoProcessControl".Robot_2.ScanNGPutFlag
              R    #ioPM_Inface.ProcessComplete
              S    #ioPM_Inface.ProcessStart
   END_STEP
   TRANSITION Trans629 FROM ScanNGPut TO ScanNGPutProcess   // T120, jump
      := "AutoProcessControl".Robot_2.ScanNGPutFlag;
   END_TRANSITION
   STEP GluePick:   // S140, max time T#10S, warning time T#7S
              S    "AutoProcessControl".Robot_2.GluePickFlag
              R    #ioPM_Inface.ProcessComplete
              S    #ioPM_Inface.ProcessStart
   END_STEP
   TRANSITION Trans638 FROM GluePick TO GluePickProcess   // T140, jump
      := "AutoProcessControl".Robot_2.GluePickFlag;
   END_TRANSITION
   STEP ScanMagane:   // S135, max time T#10S, warning time T#7S
              S    "AutoProcessControl".Robot_2.MagnetScanFlag
              R    #ioPM_Inface.ProcessComplete
              S    #ioPM_Inface.ProcessStart
   END_STEP
   TRANSITION Trans634 FROM ScanMagane TO ScanMaganeProcess   // T135, jump
      := "AutoProcessControl".Robot_2.MagnetScanFlag;
   END_TRANSITION
   STEP GlueNGPut:   // S125, max time T#10S, warning time T#7S
              S    "AutoProcessControl".Robot_2.GlueNGPutFlag
              R    #ioPM_Inface.ProcessComplete
              S    #ioPM_Inface.ProcessStart
   END_STEP
   TRANSITION Trans636 FROM GlueNGPut TO GlueNGPutProcess   // T125, jump
      := "AutoProcessControl".Robot_2.GlueNGPutFlag;
   END_TRANSITION
   STEP PickPallet:   // S115, max time T#10S, warning time T#7S
              S    "AutoProcessControl".Robot_2.PalletPickFlag
              R    #ioPM_Inface.ProcessComplete
              S    #ioPM_Inface.ProcessStart
   END_STEP
   TRANSITION Trans627 FROM PickPallet TO PickPalletProcess   // T115, jump
      := "AutoProcessControl".Robot_2.PalletPickFlag;
   END_TRANSITION
   STEP PutPress:   // S145, max time T#10S, warning time T#7S
              S    "AutoProcessControl".Robot_2.Press2PutFlag
              R    #ioPM_Inface.ProcessComplete
              S    #ioPM_Inface.ProcessStart
   END_STEP
   TRANSITION Trans639 FROM PutPress TO PutPressProcess   // T145, jump
      := "AutoProcessControl".Robot_2.Press2PutFlag;
   END_TRANSITION
   STEP Grip1SensorError:   // S266, max time T#10S, warning time T#7S
          S1  S    "ST10_DeviceError".F.Robot_2.Grip1SensorCheckError
   END_STEP
   TRANSITION Trans268 FROM Grip1SensorError TO RobotTaskSelect   // T268, jump
      := #iSysInface.Reset;
   END_TRANSITION
   STEP Grip2SensorError:   // S267, max time T#10S, warning time T#7S
          S1  S    "ST10_DeviceError".F.Robot_2.Grip2SensorCheckError
   END_STEP
   TRANSITION Trans270 FROM Grip2SensorError TO RobotTaskSelect   // T270, jump
      := #iSysInface.Reset;
   END_TRANSITION
   STEP PressPick:   // S150, max time T#10S, warning time T#7S
              R    #ioPM_Inface.ProcessComplete
              S    #ioPM_Inface.ProcessStart
   END_STEP
   TRANSITION Trans641 FROM PressPick TO PressPickProcess   // T150, jump
      := TRUE;
   END_TRANSITION
   STEP GluePut:   // S155, max time T#10S, warning time T#7S
              S    "AutoProcessControl".Robot_2.GluePutFlag
              R    #ioPM_Inface.ProcessComplete
              S    #ioPM_Inface.ProcessStart
   END_STEP
   TRANSITION Trans649 FROM GluePut TO GluePutProcess   // T155, jump
      := "AutoProcessControl".Robot_2.GluePutFlag;
   END_TRANSITION
   STEP FlagReset:   // S268, max time T#10S, warning time T#7S
              R    "AutoProcessControl".Robot_2.PalletPickFlag
              R    "AutoProcessControl".Robot_2.MagnetScanFlag
              R    "AutoProcessControl".Robot_2.GluePutFlag
              R    "AutoProcessControl".Robot_2.GluePickFlag
              R    "AutoProcessControl".Robot_2.Press2PutFlag
              R    "AutoProcessControl".Robot_2.GlueNGPutFlag
              R    "AutoProcessControl".Robot_2.ScanNGPutFlag
   END_STEP
   TRANSITION Trans271 FROM FlagReset TO "Open NG BOX REQUESTED?"   // T271
      := NOT "AutoProcessControl".Robot_2.PalletPickFlag AND NOT "AutoProcessControl".Robot_2.MagnetScanFlag AND NOT "AutoProcessControl".Robot_2.GluePutFlag AND NOT "AutoProcessControl".Robot_2.GluePickFlag AND NOT "AutoProcessControl".Robot_2.Press2PutFlag AND NOT "AutoProcessControl".Robot_2.GlueNGPutFlag AND NOT "AutoProcessControl".Robot_2.ScanNGPutFlag;
   END_TRANSITION
   STEP Maintenance:   // S131, max time T#10S, warning time T#7S
              R    #ioPM_Inface.ProcessComplete
              S    #ioPM_Inface.ProcessStart
   END_STEP
   TRANSITION Trans710 FROM Maintenance TO "Maintenance Pos"   // T131, jump
      := TRUE;
   END_TRANSITION
   STEP Masref_test:   // S132, max time T#10S, warning time T#7S
              R    #ioPM_Inface.ProcessComplete
              S    #ioPM_Inface.ProcessStart
   END_STEP
   TRANSITION Trans712 FROM Masref_test TO MasteringTest_Req   // T132, jump
      := TRUE;
   END_TRANSITION
   STEP Brake_Test:   // S133, max time T#10S, warning time T#7S
              R    #ioPM_Inface.ProcessComplete
              S    #ioPM_Inface.ProcessStart
   END_STEP
   TRANSITION Trans713 FROM Brake_Test TO BrakeTest_Req   // T133, jump
      := TRUE;
   END_TRANSITION
   STEP "Open NG BOX REQUESTED?":   // S111, max time T#10S, warning time T#7S
   END_STEP
   TRANSITION "NG BOX CLOSED" FROM "Open NG BOX REQUESTED?" TO RobotTaskSelect   // T111
      := NOT "NG_BOXES_DB".out_Request_to_open;
   END_TRANSITION

   // sequencer 3: S200-S249 Fixturecode reading
   STEP "Tablecode Scan":   // S200, max time T#10S, warning time T#7S
              R    "KukaRobot2_CtrlDB".sPLCtoROB.User.Cycle.DI307_ScanPartFinish
              R    "KukaRobot2_CtrlDB".sPLCtoROB.User.Cycle.DI306_ScanPartComplete
              N    "AutoProcessData".GripperCode_R2[1]:=''
              N    "AutoProcessData".GripperCode_R2[2]:=''
              N    "AutoProcessData".GripperCode_R2[3]:=''
              N    "AutoProcessData".GripperCode_R2[4]:=''
   END_STEP
   TRANSITION Trans147 FROM "Tablecode Scan" TO StartRobotScanGripperCode   // T200
      := TRUE;
   END_TRANSITION
   STEP "Tablecode ScanFinish":   // S149, max time T#10S, warning time T#7S
              S    #ioPM_Inface.ProcessComplete
              R    #ioPM_Inface.ProcessStart
   END_STEP
   TRANSITION Trans352 FROM "Tablecode ScanFinish" TO ProcessStart   // T149, jump
      := "ChangeOver_DB".Global.AllFixtureScanCompareOk OR "ChangeOver_DB".Robot_2.Req_RobotToMaintenancePos;
   END_TRANSITION
   STEP SetGripCodeScanFlag:   // S336, max time T#10S, warning time T#7S
   END_STEP
   TRANSITION Trans651 FROM SetGripCodeScanFlag TO "Tablecode ScanFinish"   // T623
      := TRUE;
   END_TRANSITION
   STEP WaitGripperPos1ScanFinish:   // S296, max time T#10S, warning time T#7S
   END_STEP
   TRANSITION Trans313 FROM WaitGripperPos1ScanFinish TO RobotScanGripPos1Comp   // T355
      := "KukaRobot2_CtrlDB".sPLCtoROB.User.Cycle.DI306_ScanPartComplete;
   END_TRANSITION
   STEP RobotScanGripPos1Comp:   // S301, max time T#10S, warning time T#7S
   END_STEP
   TRANSITION Trans314 FROM RobotScanGripPos1Comp TO WaitRobotScanGripPos2Reach   // T359
      := NOT "KukaRobot2_CtrlDB".sROBtoPLC.User.Cycle.DO307_ScanPos1Reach;
   END_TRANSITION
   STEP WaitRobotScanGripPos2Reach:   // S304, max time T#10S, warning time T#7S
   END_STEP
   TRANSITION Trans316 FROM WaitRobotScanGripPos2Reach TO WaitGripperPos2ScanFinish   // T360
      := "KukaRobot2_CtrlDB".sROBtoPLC.User.Cycle.DO308_ScanPos2Reach;
   END_TRANSITION
   STEP WaitGripperPos2ScanFinish:   // S337, max time T#10S, warning time T#7S
   END_STEP
   TRANSITION Trans652 FROM WaitGripperPos2ScanFinish TO RobotScanGripPos2Comp   // T626
      := "KukaRobot2_CtrlDB".sPLCtoROB.User.Cycle.DI306_ScanPartComplete;
   END_TRANSITION
   STEP RobotScanGripPos2Comp:   // S371, max time T#10S, warning time T#7S
   END_STEP
   TRANSITION Trans319 FROM RobotScanGripPos2Comp TO WaitRobotScanGripPos3Reach   // T367
      := NOT "KukaRobot2_CtrlDB".sROBtoPLC.User.Cycle.DO308_ScanPos2Reach;
   END_TRANSITION
   STEP WaitRobotScanGripPos3Reach:   // S372, max time T#10S, warning time T#7S
   END_STEP
   TRANSITION Trans320 FROM WaitRobotScanGripPos3Reach TO WaitGripperPos3ScanFinish   // T368
      := "KukaRobot2_CtrlDB".sROBtoPLC.User.Cycle.DO309_ScanPos3Reach;
   END_TRANSITION
   STEP WaitGripperPos3ScanFinish:   // S373, max time T#10S, warning time T#7S
   END_STEP
   TRANSITION Trans673 FROM WaitGripperPos3ScanFinish TO RobotScanGripPos3Comp   // T630
      := "KukaRobot2_CtrlDB".sPLCtoROB.User.Cycle.DI306_ScanPartComplete;
   END_TRANSITION
   STEP RobotScanGripPos3Comp:   // S378, max time T#10S, warning time T#7S
   END_STEP
   TRANSITION Trans323 FROM RobotScanGripPos3Comp TO WaitRobotScanGripPos4Reach   // T375
      := NOT "KukaRobot2_CtrlDB".sROBtoPLC.User.Cycle.DO309_ScanPos3Reach;
   END_TRANSITION
   STEP WaitRobotScanGripPos4Reach:   // S383, max time T#10S, warning time T#7S
   END_STEP
   TRANSITION Trans324 FROM WaitRobotScanGripPos4Reach TO WaitGripperPos4ScanFinish   // T376
      := "KukaRobot2_CtrlDB".sROBtoPLC.User.Cycle.DO310_ScanPos4Reach;
   END_TRANSITION
   STEP WaitGripperPos4ScanFinish:   // S385, max time T#10S, warning time T#7S
   END_STEP
   TRANSITION Trans676 FROM WaitGripperPos4ScanFinish TO RobotScanGripPos4Comp   // T635
      := "KukaRobot2_CtrlDB".sPLCtoROB.User.Cycle.DI306_ScanPartComplete;
   END_TRANSITION
   STEP RobotScanGripPos4Comp:   // S391, max time T#10S, warning time T#7S
              N    "KukaRobot2_CtrlDB".sPLCtoROB.User.Cycle.DI307_ScanPartFinish
              N    "KukaRobot2_CtrlDB".sPLCtoROB.User.Cycle.DI306_ScanPartComplete
   END_STEP
   TRANSITION Trans328 FROM RobotScanGripPos4Comp TO SetGripCodeScanFlag   // T383
      := "KukaRobot2_CtrlDB".sROBtoPLC.User.Cycle.DO306_GripScanFinish;
   END_TRANSITION
   STEP StartRobotScanGripperCode:   // S338, max time T#10S, warning time T#7S
              N    "KukaRobot2_CtrlDB".sPLCtoROB.User.Cycle.DI305_GripScan
   END_STEP
   TRANSITION Trans684 FROM StartRobotScanGripperCode TO RobotScanGripperReachPos1   // T616
      := "KukaRobot2_CtrlDB".sROBtoPLC.User.Cycle.DO305_GripScanInside AND NOT "KukaRobot2_CtrlDB".sROBtoPLC.User.Cycle.DO306_GripScanFinish;
   END_TRANSITION
   STEP RobotScanGripperReachPos1:   // S340, max time T#10S, warning time T#7S
   END_STEP
   TRANSITION Trans685 FROM RobotScanGripperReachPos1 TO WaitGripperPos1ScanFinish   // T673
      := "KukaRobot2_CtrlDB".sROBtoPLC.User.Cycle.DO307_ScanPos1Reach;
   END_TRANSITION

   // sequencer 4: S250-S299 PickPallet
   STEP PickPalletProcess:   // S250, max time T#10S, warning time T#7S
   END_STEP
   TRANSITION Trans150 FROM PickPalletProcess TO DataClear   // T250
      := TRUE;
   END_TRANSITION
   STEP StartRobotPickPalletShaft:   // S326, max time T#10S, warning time T#7S
              N    "KukaRobot2_CtrlDB".sPLCtoROB.User.Cycle.DI241_PickPalletReq
   END_STEP
   TRANSITION Trans607 FROM StartRobotPickPalletShaft TO WaitRobotGripHaveStatus   // T648
      := "KukaRobot2_CtrlDB".sROBtoPLC.User.Cycle.DO241_PickPalletInside AND NOT "KukaRobot2_CtrlDB".sROBtoPLC.User.Cycle.DO242_PickPalletFinish;
   END_TRANSITION
   STEP WaitRobotFinish:   // S327, max time T#10S, warning time T#7S
   END_STEP
   TRANSITION P8 FROM WaitRobotFinish TO PickPalletFinish   // T327
      := "KukaRobot2_CtrlDB".sROBtoPLC.User.Cycle.DO242_PickPalletFinish;
   END_TRANSITION
   STEP PickPalletFinish:   // S299, max time T#10S, warning time T#7S
              S    #ioPM_Inface.ProcessComplete
              R    #ioPM_Inface.ProcessStart
   END_STEP
   TRANSITION Trans654 FROM PickPalletFinish TO ProcessStart   // T299, jump
      := TRUE;
   END_TRANSITION
   STEP WaitRobotGripHaveStatus:   // S346, max time T#10S, warning time T#7S
   END_STEP
   TRANSITION Trans655 FROM WaitRobotGripHaveStatus TO Grip1PartStatus   // T655
      := ("KukaRobot2_CtrlDB".sROBtoPLC.User.Public.GO6_RobGrip2Status <> 0) OR "KukaRobot2_CtrlDB".sROBtoPLC.User.Cycle.DO242_PickPalletFinish;
   END_TRANSITION
   STEP Grip1PartStatus:   // S243, max time T#10S, warning time T#7S
      interlock C := NOT "iF-ROOBT2Gripper2CylinderInWP" AND NOT "iF-ROOBT2Gripper2CylinderInHP";
      (C)     N    "AutoProcessData".F_Robot2Grip2.PartStatus:=100
   END_STEP
   TRANSITION Trans243 FROM Grip1PartStatus TO WaitRobotFinish   // T243
      := ("iF-ROOBT2Gripper2Detection" AND ("AutoProcessData".F_Robot2Grip2.PartStatus = 100)) OR (NOT "iF-ROOBT2Gripper2Detection" AND (#Grip1PartStatus.T > t#500MS));
   END_TRANSITION
   STEP DataClear:   // S252, max time T#10S, warning time T#7S
          S1  N    "AutoProcessData".F_Robot2Grip2:="AutoProcessData".ClearData
   END_STEP
   TRANSITION Trans253 FROM DataClear TO StartRobotPickPalletShaft   // T253
      := TRUE;
   END_TRANSITION

   // sequencer 5: S300-S349 ScanNGPut
   STEP ScanNGPutProcess:   // S300, max time T#10S, warning time T#7S
   END_STEP
   TRANSITION Trans300 FROM ScanNGPutProcess TO StartRobotScanNGPut   // T300
      := TRUE;
   END_TRANSITION
   STEP DataMove:   // S253, max time T#10S, warning time T#7S
          S1  N    "AutoProcessData".C_MagnScanNGBuffer:="AutoProcessData".F_Robot2Grip2
          S1  N    "AutoProcessData".F_Robot2Grip2:="AutoProcessData".ClearData
   END_STEP
   TRANSITION Trans254 FROM DataMove TO WaitRobotFinish_1   // T254
      := #DataMove.T > t#100MS;
   END_TRANSITION
   STEP StartRobotScanNGPut:   // S328, max time T#10S, warning time T#7S
              N    "KukaRobot2_CtrlDB".sPLCtoROB.User.Cycle.DI249_ScanNGPutReq
   END_STEP
   TRANSITION Trans610 FROM StartRobotScanNGPut TO WaitRobotGripHaveStatus_1   // T328
      := "KukaRobot2_CtrlDB".sROBtoPLC.User.Cycle.DO249_ScanNGPutInside AND NOT "KukaRobot2_CtrlDB".sROBtoPLC.User.Cycle.DO250_ScanNGPutFinish;
   END_TRANSITION
   STEP WaitRobotFinish_1:   // S343, max time T#10S, warning time T#7S
   END_STEP
   TRANSITION P9 FROM WaitRobotFinish_1 TO ScanNGPutFinish_1   // T651
      := "KukaRobot2_CtrlDB".sROBtoPLC.User.Cycle.DO250_ScanNGPutFinish AND "iE-NG-03MagnetDispenseNGDetection" AND (#WaitRobotFinish_1.T > t#100MS);
   END_TRANSITION
   TRANSITION Trans930 FROM WaitRobotFinish_1 TO Step930   // T930
      := "KukaRobot2_CtrlDB".sROBtoPLC.User.Cycle.DO250_ScanNGPutFinish AND NOT "iE-NG-03MagnetDispenseNGDetection" AND "ST10Cylinder".Cy[16].In.HomePositionSensor AND (#WaitRobotFinish_1.T > t#5S);
   END_TRANSITION
   STEP ScanNGPutFinish_1:   // S349, max time T#10S, warning time T#7S
              S    #ioPM_Inface.ProcessComplete
              R    #ioPM_Inface.ProcessStart
   END_STEP
   TRANSITION Trans656 FROM ScanNGPutFinish_1 TO ProcessStart   // T349, jump
      := TRUE;
   END_TRANSITION
   STEP WaitRobotGripHaveStatus_1:   // S347, max time T#10S, warning time T#7S
   END_STEP
   TRANSITION Trans657 FROM WaitRobotGripHaveStatus_1 TO DataMove   // T656
      := "KukaRobot2_CtrlDB".sROBtoPLC.User.Public.GO6_RobGrip2Status = 0;
   END_TRANSITION
   STEP Step930:   // S930, max time T#10S, warning time T#7S
              N    "AutoProcessData".C_MagnScanNGBuffer.PartStatus:=0
   END_STEP
   TRANSITION Trans931 FROM Step930 TO ProcessStart   // T931, jump
      := #Step930.T > t#100MS;
   END_TRANSITION

   // sequencer 6: S350-S399 GlueNGPut
   STEP GlueNGPutProcess:   // S350, max time T#10S, warning time T#7S
   END_STEP
   TRANSITION Trans350 FROM GlueNGPutProcess TO StartRobotGlueNGPut   // T350
      := TRUE;
   END_TRANSITION
   STEP DataMove_1:   // S255, max time T#10S, warning time T#7S
          S1  N    "AutoProcessData".C_GlueNGBuffer:="AutoProcessData".F_Robot2Grip1
          S1  N    "AutoProcessData".F_Robot2Grip1:="AutoProcessData".ClearData
   END_STEP
   TRANSITION Trans256 FROM DataMove_1 TO WaitRobotFinish_2   // T256
      := #DataMove_1.T > t#100MS;
   END_TRANSITION
   STEP StartRobotGlueNGPut:   // S344, max time T#10S, warning time T#7S
              N    "KukaRobot2_CtrlDB".sPLCtoROB.User.Cycle.DI253_GlueNGPutReq
   END_STEP
   TRANSITION Trans611 FROM StartRobotGlueNGPut TO WaitRobotGripHaveStatus_2   // T652
      := "KukaRobot2_CtrlDB".sROBtoPLC.User.Cycle.DO253_GlueNGPutInside AND NOT "KukaRobot2_CtrlDB".sROBtoPLC.User.Cycle.DO254_GlueNGPutFinish;
   END_TRANSITION
   STEP WaitRobotFinish_2:   // S345, max time T#10S, warning time T#7S
   END_STEP
   TRANSITION P10 FROM WaitRobotFinish_2 TO GlueNGPutFinish   // T653
      := "KukaRobot2_CtrlDB".sROBtoPLC.User.Cycle.DO254_GlueNGPutFinish;
   END_TRANSITION
   STEP GlueNGPutFinish:   // S399, max time T#10S, warning time T#7S
              S    #ioPM_Inface.ProcessComplete
              R    #ioPM_Inface.ProcessStart
   END_STEP
   TRANSITION Trans658 FROM GlueNGPutFinish TO ProcessStart   // T399, jump
      := TRUE;
   END_TRANSITION
   STEP WaitRobotGripHaveStatus_2:   // S348, max time T#10S, warning time T#7S
   END_STEP
   TRANSITION Trans659 FROM WaitRobotGripHaveStatus_2 TO DataMove_1   // T657
      := "KukaRobot2_CtrlDB".sROBtoPLC.User.Public.GO5_RobGrip1Status = 0;
   END_TRANSITION

   // sequencer 7: S400-S449 PickTable
   STEP PickTableProcess:   // S400, max time T#10S, warning time T#7S
   END_STEP
   TRANSITION Trans400 FROM PickTableProcess TO "Data Clear_2"   // T400
      := TRUE;
   END_TRANSITION
   STEP Grip2PartStatus:   // S244, max time T#10S, warning time T#7S
              N    "AutoProcessData".F_Robot2Grip2.PartStatus:=100
   END_STEP
   TRANSITION Trans244 FROM Grip2PartStatus TO WaitRobotFinish_3   // T244
      := "AutoProcessData".F_Robot2Grip2.PartStatus = 100;
   END_TRANSITION
   STEP StartRobotPickTable:   // S352, max time T#10S, warning time T#7S
              N    "KukaRobot2_CtrlDB".sPLCtoROB.User.Cycle.DI257_PickPartReq
   END_STEP
   TRANSITION Trans618 FROM StartRobotPickTable TO WaitRobotGripHaveStatus_3   // T654
      := "KukaRobot2_CtrlDB".sROBtoPLC.User.Cycle.DO257_PickPartInside AND NOT "KukaRobot2_CtrlDB".sROBtoPLC.User.Cycle.DO258_PickPartFinish;
   END_TRANSITION
   STEP WaitRobotFinish_3:   // S353, max time T#10S, warning time T#7S
   END_STEP
   TRANSITION P11 FROM WaitRobotFinish_3 TO PickTableProcessFinish   // T658
      := "KukaRobot2_CtrlDB".sROBtoPLC.User.Cycle.DO258_PickPartFinish;
   END_TRANSITION
   STEP PickTableProcessFinish:   // S449, max time T#10S, warning time T#7S
              S    #ioPM_Inface.ProcessComplete
              R    #ioPM_Inface.ProcessStart
   END_STEP
   TRANSITION Trans660 FROM PickTableProcessFinish TO ProcessStart   // T449, jump
      := TRUE;
   END_TRANSITION
   STEP WaitRobotGripHaveStatus_3:   // S354, max time T#10S, warning time T#7S
   END_STEP
   TRANSITION Trans661 FROM WaitRobotGripHaveStatus_3 TO Grip2PartStatus   // T659
      := "KukaRobot2_CtrlDB".sROBtoPLC.User.Public.GO6_RobGrip2Status <> 0;
   END_TRANSITION
   STEP "Data Clear_2":   // S258, max time T#10S, warning time T#7S
          S1  N    "AutoProcessData".F_Robot2Grip2:="AutoProcessData".ClearData
   END_STEP
   TRANSITION Trans259 FROM "Data Clear_2" TO StartRobotPickTable   // T259
      := #"Data Clear_2".T > t#100MS;
   END_TRANSITION

   // sequencer 8: S450-S499 ScanMagane
   STEP ScanMaganeProcess:   // S450, max time T#10S, warning time T#7S
   END_STEP
   TRANSITION Trans450 FROM ScanMaganeProcess TO StartRobotScanRing   // T450
      := TRUE;
   END_TRANSITION
   STEP CheckScanReady:   // S245, max time T#10S, warning time T#7S
   END_STEP
   TRANSITION Trans245 FROM CheckScanReady TO ScanStart   // T245
      := "KeyenceSR1000Ctrl_806A1DB".oReady;
   END_TRANSITION
   STEP StartRobotScanRing:   // S355, max time T#10S, warning time T#7S
              N    "KukaRobot2_CtrlDB".sPLCtoROB.User.Cycle.DI261_ScanPartReq
   END_STEP
   TRANSITION Trans619 FROM StartRobotScanRing TO WaitRobotReachScanPos   // T660
      := "KukaRobot2_CtrlDB".sROBtoPLC.User.Cycle.DO261_ScanPartInside AND NOT "KukaRobot2_CtrlDB".sROBtoPLC.User.Cycle.DO262_ScanPartFinish;
   END_TRANSITION
   STEP WaitRobotFinish_4:   // S356, max time T#10S, warning time T#7S
              N    "KukaRobot2_CtrlDB".sPLCtoROB.User.Cycle.DI262_ScanPartComplete
   END_STEP
   TRANSITION P12 FROM WaitRobotFinish_4 TO ScanMaganeProcessFinish   // T661
      := "KukaRobot2_CtrlDB".sROBtoPLC.User.Cycle.DO262_ScanPartFinish;
   END_TRANSITION
   STEP ScanMaganeProcessFinish:   // S499, max time T#10S, warning time T#7S
              S    #ioPM_Inface.ProcessComplete
              R    #ioPM_Inface.ProcessStart
   END_STEP
   TRANSITION Trans662 FROM ScanMaganeProcessFinish TO ProcessStart   // T499, jump
      := TRUE;
   END_TRANSITION
   STEP WaitRobotReachScanPos:   // S357, max time T#10S, warning time T#7S
   END_STEP
   TRANSITION Trans663 FROM WaitRobotReachScanPos TO CheckScanReady   // T662
      := "KukaRobot2_CtrlDB".sROBtoPLC.User.Cycle.DO263_ScanReach;
   END_TRANSITION
   STEP ScanStart:   // S246, max time T#10S, warning time T#7S
          S1  S    "KeyenceSR1000Ctrl_806A1DB".ioAutoTrigger
   END_STEP
   TRANSITION Trans246 FROM ScanStart TO WaitScanCompletely   // T246
      := NOT "KeyenceSR1000Ctrl_806A1DB".sHMI.Status.Ready;
   END_TRANSITION
   STEP WaitScanCompletely:   // S247, max time T#10S, warning time T#7S
   END_STEP
   TRANSITION Trans247 FROM WaitScanCompletely TO CodeMove   // T247
      := "KeyenceSR1000Ctrl_806A1DB".sHMI.Status.Complete AND "KeyenceSR1000Ctrl_806A1DB".sHMI.Status.ReadOk;
   END_TRANSITION
   TRANSITION Trans248 FROM WaitScanCompletely TO PartNGStatus   // T248
      := "KeyenceSR1000Ctrl_806A1DB".sHMI.Status.Complete AND "KeyenceSR1000Ctrl_806A1DB".sHMI.Status.ReadNok;
   END_TRANSITION
   STEP CodeMove:   // S248, max time T#10S, warning time T#7S
              N    "AutoProcessData".F_Robot2Grip2.Code_1:="KeyenceSR1000Ctrl_806A1DB".sHMI.Status.CurrentCode
   END_STEP
   TRANSITION Trans249 FROM CodeMove TO PartOKStatus_1   // T249
      := TRUE;
   END_TRANSITION
   STEP PartOKStatus:   // S249, max time T#10S, warning time T#7S
              N    "AutoProcessData".F_Robot2Grip2.PartStatus:=199
   END_STEP
   TRANSITION Trans251 FROM PartOKStatus TO WaitRobotFinish_4   // T251
      := "AutoProcessData".F_Robot2Grip2.PartStatus = 199;
   END_TRANSITION
   STEP PartNGStatus:   // S251, max time T#10S, warning time T#7S
              N    "AutoProcessData".F_Robot2Grip2.PartStatus:=155
   END_STEP
   TRANSITION Trans252 FROM PartNGStatus TO WaitRobotFinish_4   // T252
      := "AutoProcessData".F_Robot2Grip2.PartStatus = 155;
   END_TRANSITION
   STEP PartOKStatus_1:   // S269, max time T#10S, warning time T#7S
              N    "AutoProcessData".F_Robot2Grip2.PartStatus:=110
   END_STEP
   TRANSITION Trans272 FROM PartOKStatus_1 TO "MES Online  offline?"   // T272
      := "AutoProcessData".F_Robot2Grip2.PartStatus = 110;
   END_TRANSITION
   STEP "MES Online  offline?":   // S384, max time T#10S, warning time T#7S
   END_STEP
   TRANSITION Offline FROM "MES Online  offline?" TO PartOKStatus   // T698
      := "Station_Sys".Cmd.OnOffLine;
   END_TRANSITION
   TRANSITION Trans700 FROM "MES Online  offline?" TO WaitRobotFinish_4   // T700
      := NOT "Station_Sys".Cmd.OnOffLine;
   END_TRANSITION

   // sequencer 9: S500-S549 GluePick
   STEP GluePickProcess:   // S500, max time T#10S, warning time T#7S
   END_STEP
   TRANSITION Trans500 FROM GluePickProcess TO StartRobotGluePick   // T500
      := TRUE;
   END_TRANSITION
   STEP DataMove_2:   // S257, max time T#10S, warning time T#7S
          S1  N    "AutoProcessData".F_Robot2Grip1:="AutoProcessData".C_Glue
          S1  N    "AutoProcessData".C_Glue:="AutoProcessData".ClearData
   END_STEP
   TRANSITION Trans258 FROM DataMove_2 TO WaitRobotFinish_5   // T258
      := #DataMove_2.T > t#100MS;
   END_TRANSITION
   STEP StartRobotGluePick:   // S358, max time T#10S, warning time T#7S
              N    "KukaRobot2_CtrlDB".sPLCtoROB.User.Cycle.DI269_GluePickReq
   END_STEP
   TRANSITION Trans646 FROM StartRobotGluePick TO WaitRobotGripStatus   // T663
      := "KukaRobot2_CtrlDB".sROBtoPLC.User.Cycle.DO269_GluePickInside AND NOT "KukaRobot2_CtrlDB".sROBtoPLC.User.Cycle.DO270_GluePickFinish;
   END_TRANSITION
   STEP WaitRobotFinish_5:   // S359, max time T#10S, warning time T#7S
   END_STEP
   TRANSITION P13 FROM WaitRobotFinish_5 TO PressGluePickProcessFinish   // T664
      := "KukaRobot2_CtrlDB".sROBtoPLC.User.Cycle.DO270_GluePickFinish;
   END_TRANSITION
   STEP PressGluePickProcessFinish:   // S549, max time T#10S, warning time T#7S
              S    #ioPM_Inface.ProcessComplete
              R    #ioPM_Inface.ProcessStart
   END_STEP
   TRANSITION Trans664 FROM PressGluePickProcessFinish TO ProcessStart   // T549, jump
      := TRUE;
   END_TRANSITION
   STEP WaitRobotGripStatus:   // S360, max time T#10S, warning time T#7S
   END_STEP
   TRANSITION Trans665 FROM WaitRobotGripStatus TO DataMove_2   // T665
      := "KukaRobot2_CtrlDB".sROBtoPLC.User.Public.GO5_RobGrip1Status <> 0;
   END_TRANSITION

   // sequencer 10: S550-S599 PutPress
   STEP PutPressProcess:   // S550, max time T#10S, warning time T#7S
   END_STEP
   TRANSITION Trans550 FROM PutPressProcess TO StartRobotPutPress   // T550
      := TRUE;
   END_TRANSITION
   STEP DataMove_3:   // S260, max time T#10S, warning time T#7S
          S1  N    "AutoProcessData".B_Press2:="AutoProcessData".F_Robot2Grip1
          S1  N    "AutoProcessData".F_Robot2Grip1:="AutoProcessData".ClearData
   END_STEP
   TRANSITION Trans261 FROM DataMove_3 TO WaitRobotFinish_6   // T261
      := #DataMove_3.T > t#100MS;
   END_TRANSITION
   STEP StartRobotPutPress:   // S361, max time T#10S, warning time T#7S
              N    "KukaRobot2_CtrlDB".sPLCtoROB.User.Cycle.DI273_PutPressReq
   END_STEP
   TRANSITION Trans647 FROM StartRobotPutPress TO WaitRobotGripStatus_1   // T666
      := "KukaRobot2_CtrlDB".sROBtoPLC.User.Cycle.DO273_PressPutPart1Inside AND NOT "KukaRobot2_CtrlDB".sROBtoPLC.User.Cycle.DO274_PressPutPart1Finish;
   END_TRANSITION
   STEP WaitRobotFinish_6:   // S362, max time T#10S, warning time T#7S
   END_STEP
   TRANSITION P14 FROM WaitRobotFinish_6 TO PutProcessFinish   // T667
      := "KukaRobot2_CtrlDB".sROBtoPLC.User.Cycle.DO274_PressPutPart1Finish;
   END_TRANSITION
   STEP PutProcessFinish:   // S599, max time T#10S, warning time T#7S
              S    #ioPM_Inface.ProcessComplete
              R    #ioPM_Inface.ProcessStart
              N    "Robot_DB".Robot_2.SpeedCount:="Robot_DB".Robot_2.SpeedCount+1
   END_STEP
   TRANSITION Trans666 FROM PutProcessFinish TO ProcessStart   // T599, jump
      := TRUE;
   END_TRANSITION
   STEP WaitRobotGripStatus_1:   // S363, max time T#10S, warning time T#7S
   END_STEP
   TRANSITION Trans667 FROM WaitRobotGripStatus_1 TO DataMove_3   // T668
      := "KukaRobot2_CtrlDB".sROBtoPLC.User.Public.GO5_RobGrip1Status = 0;
   END_TRANSITION

   // sequencer 11: S600-S649 PressPick
   STEP PressPickProcess:   // S600, max time T#10S, warning time T#7S
   END_STEP
   TRANSITION Trans600 FROM PressPickProcess TO StartRobotPressPick   // T600
      := TRUE;
   END_TRANSITION
   STEP DataMove_4:   // S262, max time T#10S, warning time T#7S
          S1  N    "AutoProcessData".F_Robot2Grip1:="AutoProcessData".B_Press1
          S1  N    "AutoProcessData".B_Press1:="AutoProcessData".ClearData
   END_STEP
   TRANSITION Trans263 FROM DataMove_4 TO WaitRobotFinish_7   // T263
      := #DataMove_4.T > t#100MS;
   END_TRANSITION
   STEP StartRobotPressPick:   // S364, max time T#10S, warning time T#7S
   END_STEP
   TRANSITION Trans648 FROM StartRobotPressPick TO WaitRobotGripStatus_2   // T669
      := "AlwaysTRUE" AND NOT "AlwaysTRUE";
   END_TRANSITION
   STEP WaitRobotFinish_7:   // S365, max time T#10S, warning time T#7S
   END_STEP
   TRANSITION P15 FROM WaitRobotFinish_7 TO PressPickProcessFinish_   // T670
      := "AlwaysTRUE";
   END_TRANSITION
   STEP PressPickProcessFinish_:   // S649, max time T#10S, warning time T#7S
              S    #ioPM_Inface.ProcessComplete
              R    #ioPM_Inface.ProcessStart
   END_STEP
   TRANSITION Trans668 FROM PressPickProcessFinish_ TO ProcessStart   // T649, jump
      := TRUE;
   END_TRANSITION
   STEP WaitRobotGripStatus_2:   // S366, max time T#10S, warning time T#7S
   END_STEP
   TRANSITION Trans669 FROM WaitRobotGripStatus_2 TO DataMove_4   // T671
      := "KukaRobot2_CtrlDB".sROBtoPLC.User.Public.GO5_RobGrip1Status <> 0;
   END_TRANSITION

   // sequencer 12: S650-S699 GluePut
   STEP GluePutProcess:   // S650, max time T#10S, warning time T#7S
   END_STEP
   TRANSITION Trans674 FROM GluePutProcess TO StartRobotGluePut   // T650
      := TRUE;
   END_TRANSITION
   STEP DataMove_5:   // S264, max time T#10S, warning time T#7S
              N    "AutoProcessData".C_Glue.Code_1:="AutoProcessData".F_Robot2Grip2.Code_1
              N    "AutoProcessData".C_Glue.PartStatus:=320
   END_STEP
   TRANSITION Trans265 FROM DataMove_5 TO "Data Clear_6"   // T265
      := #DataMove_5.T > t#100MS;
   END_TRANSITION
   STEP StartRobotGluePut:   // S367, max time T#10S, warning time T#7S
              N    "KukaRobot2_CtrlDB".sPLCtoROB.User.Cycle.DI265_GluePutReq
   END_STEP
   TRANSITION Trans650 FROM StartRobotGluePut TO WaitRobotGripStatus_3   // T676
      := "KukaRobot2_CtrlDB".sROBtoPLC.User.Cycle.DO265_GluePutInside AND NOT "KukaRobot2_CtrlDB".sROBtoPLC.User.Cycle.DO266_GluePutFinish;
   END_TRANSITION
   STEP WaitRobotFinish_8:   // S368, max time T#10S, warning time T#7S
   END_STEP
   TRANSITION P16 FROM WaitRobotFinish_8 TO GluePutProcessFinish   // T677
      := "KukaRobot2_CtrlDB".sROBtoPLC.User.Cycle.DO266_GluePutFinish;
   END_TRANSITION
   STEP GluePutProcessFinish:   // S699, max time T#10S, warning time T#7S
              S    #ioPM_Inface.ProcessComplete
              R    #ioPM_Inface.ProcessStart
   END_STEP
   TRANSITION Trans670 FROM GluePutProcessFinish TO ProcessStart   // T699, jump
      := TRUE;
   END_TRANSITION
   STEP WaitRobotGripStatus_3:   // S369, max time T#10S, warning time T#7S
   END_STEP
   TRANSITION Trans671 FROM WaitRobotGripStatus_3 TO DataMove_5   // T679
      := "KukaRobot2_CtrlDB".sROBtoPLC.User.Public.GO6_RobGrip2Status = 0;
   END_TRANSITION
   STEP "Data Clear_6":   // S265, max time T#10S, warning time T#7S
          S1  N    "AutoProcessData".F_Robot2Grip2:="AutoProcessData".ClearData
   END_STEP
   TRANSITION Trans266 FROM "Data Clear_6" TO WaitRobotFinish_8   // T266
      := TRUE;
   END_TRANSITION

   // sequencer 13: S850-S899 Maintenance Pos
   STEP "Maintenance Pos":   // S850, max time T#10S, warning time T#7S
   END_STEP
   TRANSITION Trans704 FROM "Maintenance Pos" TO ReqRobotToMantenPos_1   // T850
      := "KukaRobot3_CtrlDB".sROBtoPLC.User.Cycle.DO298_MaintainFinish OR "KukaRobot3_CtrlDB".sROBtoPLC.Sys.SO.IN_HOME;
   END_TRANSITION
   STEP ReqRobotToMantenPos_1:   // S704, max time T#10S, warning time T#7S
              N    "KukaRobot2_CtrlDB".sPLCtoROB.User.Cycle.DI297_MaintainRequest
   END_STEP
   TRANSITION Trans705 FROM ReqRobotToMantenPos_1 TO WaitR1MaintenPosFinsh_1   // T705
      := "KukaRobot2_CtrlDB".sROBtoPLC.User.Cycle.DO297_MaintainInside AND NOT "KukaRobot2_CtrlDB".sROBtoPLC.User.Cycle.DO298_MaintainFinish;
   END_TRANSITION
   STEP WaitR1MaintenPosFinsh_1:   // S705, max time T#10S, warning time T#7S
              R    "AutoProcessControl".Robot_2.MaintenanceRequest
   END_STEP
   TRANSITION Trans706 FROM WaitR1MaintenPosFinsh_1 TO WaitRobotHomeRequest   // T706
      := NOT "KukaRobot2_CtrlDB".sROBtoPLC.User.Cycle.DO297_MaintainInside AND "KukaRobot2_CtrlDB".sROBtoPLC.User.Cycle.DO298_MaintainFinish AND NOT "AutoProcessControl".Robot_2.MaintenanceRequest AND NOT "ChangeOver_DB".Robot_2.Req_RobotToMaintenancePos;
   END_TRANSITION
   STEP WaitRobotHomeRequest:   // S706, max time T#10S, warning time T#7S
          S1  R    "ChangeOver_DB".Robot_2.MaintenancePosReqSelFlag
   END_STEP
   TRANSITION Trans707 FROM WaitRobotHomeRequest TO ReqRobotToHomePos   // T707
      := "ChangeOver_DB".Robot_2.HMI_MaintenanceHomeReq AND ("KukaRobot3_CtrlDB".sROBtoPLC.User.Cycle.DO298_MaintainFinish OR "KukaRobot3_CtrlDB".sROBtoPLC.Sys.SO.IN_HOME) AND NOT "KukaRobot2_CtrlDB".sROBtoPLC.User.Cycle.DO300_HomeInside;
   END_TRANSITION
   STEP ReqRobotToHomePos:   // S707, max time T#10S, warning time T#7S
              N    "KukaRobot2_CtrlDB".sPLCtoROB.User.Cycle.DI300_HomeRequest
   END_STEP
   TRANSITION Trans708 FROM ReqRobotToHomePos TO WaitR1HomePosFinsh_1   // T708
      := "KukaRobot2_CtrlDB".sROBtoPLC.User.Cycle.DO300_HomeInside AND NOT "KukaRobot2_CtrlDB".sROBtoPLC.User.Cycle.DO301_HomeFinish;
   END_TRANSITION
   STEP WaitR1HomePosFinsh_1:   // S899, max time T#10S, warning time T#7S
   END_STEP
   TRANSITION Trans709 FROM WaitR1HomePosFinsh_1 TO ProcessStart   // T899, jump
      := NOT "KukaRobot2_CtrlDB".sROBtoPLC.User.Cycle.DO300_HomeInside AND "KukaRobot2_CtrlDB".sROBtoPLC.User.Cycle.DO301_HomeFinish AND NOT "AutoProcessControl".Robot_2.HomeRequest;
   END_TRANSITION

   // sequencer 14: S900S950 Test
   STEP "900":   // S900, max time T#10S, warning time T#7S
   END_STEP
   TRANSITION Trans134 FROM "900" TO (MasteringTest_Req, BrakeTest_Req)   // T134
      := TRUE;
   END_TRANSITION
   STEP MasteringTest_Req:   // S910, max time T#10S, warning time T#7S
              N    "KukaRobot2_CtrlDB".sPLCtoROB.User.Cycle.DI321
              N    "KukaRobot2_CtrlDB".sPLCtoROB.User.Safety.DI450
   END_STEP
   TRANSITION Trans136 FROM MasteringTest_Req TO WaitMasteringTestFinish   // T136
      := "KukaRobot2_CtrlDB".sROBtoPLC.User.Safety.DO462;
   END_TRANSITION
   STEP BrakeTest_Req:   // S920, max time T#10S, warning time T#7S
              N    "KukaRobot2_CtrlDB".sPLCtoROB.User.Cycle.DI329
              N    "KukaRobot2_CtrlDB".sPLCtoROB.User.Safety.DI451
   END_STEP
   TRANSITION Trans138 FROM BrakeTest_Req TO WaitBrakeTestFinish   // T138
      := "KukaRobot2_CtrlDB".sROBtoPLC.User.Safety.DO453;
   END_TRANSITION
   STEP WaitMasteringTestFinish:   // S911, max time T#10S, warning time T#7S
   END_STEP
   TRANSITION Trans139 FROM WaitMasteringTestFinish TO MasteringTestFinish   // T139
      := NOT "KukaRobot2_CtrlDB".sROBtoPLC.User.Safety.DO460 AND NOT "KukaRobot2_CtrlDB".sROBtoPLC.User.Safety.DO462 AND "KukaRobot2_CtrlDB".sROBtoPLC.User.Safety.DO461;
   END_TRANSITION
   STEP WaitBrakeTestFinish:   // S921, max time T#10S, warning time T#7S
   END_STEP
   TRANSITION Trans141 FROM WaitBrakeTestFinish TO BrakeTestFinish   // T141
      := NOT "KukaRobot2_CtrlDB".sROBtoPLC.User.Safety.DO452 AND NOT "KukaRobot2_CtrlDB".sROBtoPLC.User.Safety.DO453 AND "KukaRobot2_CtrlDB".sROBtoPLC.User.Safety.DO454;
   END_TRANSITION
   STEP MasteringTestFinish:   // S919, max time T#10S, warning time T#7S
              R    "Robot_DB".Robot_2.MasteringTest_Req
   END_STEP
   TRANSITION Trans142 FROM MasteringTestFinish TO ProcessStart   // T919, jump
      := NOT "Robot_DB".Robot_2.MasteringTest_Req;
   END_TRANSITION
   STEP BrakeTestFinish:   // S929, max time T#10S, warning time T#7S
              R    "Robot_DB".Robot_2.BrakeTest_Req
   END_STEP
   TRANSITION Trans995 FROM BrakeTestFinish TO ProcessStart   // T929, jump
      := NOT "Robot_DB".Robot_2.BrakeTest_Req;
   END_TRANSITION

   // permanent post-instructions
   NETWORK 1
      #ioPM_Inface.StepNum := #RT_DATA.S_DISPLAY;
   NETWORK 2
      IF #iSysInface.Reset THEN #AlarmID := 0; END_IF;
   NETWORK 3
      #TON[10].TON(IN := #工件放行中, PT := T#0.5S);
      IF #TON[10].Q THEN #工件放行中 := FALSE; END_IF;
END_FUNCTION_BLOCK
